METHOD M_CheckGCodeStart : ERRORID
VAR_INPUT
END_VAR
IF NOT (P_bIsInit AND pDiluter^.P_bIsInit) THEN
	M_CheckGCodeStart := E_ErrorIdCmd.ERRORID_DeviceNotInitialized;
END_IF
END_METHOD

METHOD M_CheckProcDataType : BOOL
VAR_INPUT
	eProcDataType : E_ProcDataType;
END_VAR
IF eProcDataType = E_ProcDataType.PROCDATATYPE_Temp1 THEN
	M_CheckProcDataType := TRUE;
END_IF
END_METHOD

METHOD M_CheckProps : ERRORID
VAR_INPUT
END_VAR
M_CheckProps := SUPER^.M_CheckProps();
IF M_CheckProps > 0 THEN
	RETURN;
END_IF
//Konfigurierte Properties checken
//zugeordneter Diuter
IF fbObjectDirectory.M_GetObjType(nDiluterObjId) <> E_ObjectType.OBJECTTYPE_Diluter THEN
	M_CheckProps := E_ErrorIdObjMgmt.ERRORID_InvalidDiluterObjId; //Error
	RETURN;
ELSE
	pDiluter := fbObjectDirectory.M_GetObjPointer(nDiluterObjId);
END_IF
END_METHOD

METHOD M_ExeAction : ERRORID
VAR_INPUT
	refActionData : REFERENCE TO ST_ActionData;	
END_VAR
IF NOT (eCurrentState = E_MachineState.MACHINESTATE_Idle OR
	eCurrentState = E_MachineState.MACHINESTATE_Active OR
	eCurrentState = E_MachineState.MACHINESTATE_Ready) THEN
	M_ExeAction := E_ErrorIdCmd.ERRORID_InvalidState;
	RETURN;
END_IF

CASE refActionData.eAction OF
	
	E_Action.ACTION_Init:
		IF NOT bInitAxis AND NOT bInitTool THEN
			bInitAxis := TRUE;
			bInitTool := TRUE;
			fbList.A_AddHeadValue( hList := hList, putValue := E_Action.ACTION_Init);	//InitBase
			fbList.A_AddHeadValue( hList := hList, putValue := E_Action.ACTION_Init);	//InitSpec
		ELSE
			RETURN;
		END_IF		
	
	E_Action.ACTION_Heating:
		IF nStateA_Heating = 0 THEN
			nTempSetpoint := DINT_TO_UINT(refActionData.aParams[1]);
			IF nTempSetpoint > 1000 THEN
				M_ExeAction := E_ErrorIdCmd.ERRORID_InvalidHeatingTemp;  //Error
				RETURN;
			END_IF
			bHeatingOn := DINT_TO_BOOL(refActionData.aParams[2]);			
			bHeating := TRUE;
			fbList.A_AddHeadValue(hList := hList, putValue := E_Action.ACTION_Heating);
		ELSE
			RETURN;
		END_IF		
		
	E_Action.ACTION_Aspirate:
		IF NOT bAspirate THEN
			M_ExeAction := pDiluter^.M_CheckBottles(0); //Checken, ob Bottles OK
			IF M_ExeAction > 0 THEN
				RETURN;
			END_IF
			nQuantity := refActionData.aParams[1];
			nFlow := refActionData.aParams[2];
			fbList.A_AddHeadValue( hList := hList, putValue := E_Action.ACTION_Aspirate);
			bAspirate := TRUE;
		END_IF
		
	E_Action.ACTION_Dispense:
		IF NOT bDispense THEN
			M_ExeAction := pDiluter^.M_CheckBottles(0); //Checken, ob Bottles OK
			IF M_ExeAction > 0 THEN
				RETURN;
			END_IF
			nQuantity := refActionData.aParams[1];
			nFlow := refActionData.aParams[2];
			fbList.A_AddHeadValue( hList := hList, putValue := E_Action.ACTION_Dispense);
			bDispense := TRUE;
		END_IF
		
	E_Action.ACTION_DispenseDrops:
		bDispensePiezoStart := DINT_TO_BOOL(refActionData.aParams[2]);
		IF NOT bDispensePiezo AND bDispensePiezoStart THEN
			fbPiezoControl.P_nDrops := nDrops := DINT_TO_UINT(refActionData.aParams[1]);
			fbPiezoControl.P_bStroboscope := DINT_TO_BOOL(refActionData.aParams[3]);
			bSkipValveMove := DINT_TO_BOOL(refActionData.aParams[5]);
			fbList.A_AddHeadValue(hList := hList, putValue := E_Action.ACTION_DispenseDrops);
			bDispensePiezo := TRUE;
		ELSE
			fbPiezoControl.M_StartStop(bDispensePiezoStart); //Stoppen
		END_IF
		
	E_Action.ACTION_DilMoveValve:
		//Darf nur ausgeführt werden, wenn kein Dispensen aktiv ist
		IF NOT (bAspirate OR bDispense OR bDispensePiezo OR bDilMoveValve) THEN
			M_ExeAction := pDiluter^.M_ExeAction(refActionData);
			IF M_ExeAction > 0 THEN
				RETURN;
			END_IF
			fbList.A_AddHeadValue(hList := hList, putValue := E_Action.ACTION_DilMoveValve);
			bDilMoveValve := TRUE;
		END_IF
		
	E_Action.ACTION_MoveX,E_Action.ACTION_MoveY,E_Action.ACTION_MoveXY:
		IF pZAxisRef^.stInput.nToolState.1 THEN	//ZSensor ist montiert
			M_ExeAction := ERRORID_PipMoveWithZSensor;  //Error
			RETURN;
		ELSE
			M_ExeAction := SUPER^.M_ExeAction(refActionData);
			RETURN;
		END_IF

	E_Action.ACTION_MoveZ:
		IF pZAxisRef^.stInput.nToolState.1 THEN //ZSensor ist montiert
			eMoveModeZ := DINT_TO_USINT(refActionData.aParams[1]);
			IF NOT(eMoveModeZ = E_MoveMode.MODE_Free OR eMoveModeZ = E_MoveMode.MODE_Home) THEN
				M_ExeAction := ERRORID_PipMoveWithZSensor;  //Error
				RETURN;
			END_IF
			M_ExeAction := SUPER^.M_ExeAction(refActionData);
			RETURN;			
		ELSE
			M_ExeAction := SUPER^.M_ExeAction(refActionData);
			RETURN;
		END_IF
	ELSE
		M_ExeAction := SUPER^.M_ExeAction(refActionData);
		RETURN;
END_CASE
bBusy := TRUE;
eCurrentState := E_MachineState.MACHINESTATE_Active;
END_METHOD

METHOD M_GetAllProps : ERRORID
VAR_INPUT
	refCmdData : REFERENCE TO  ST_CmdData;
END_VAR
//BaseProperties lesen
SUPER^.M_GetAllProps(refCmdData);
nCurrentPropIndex := nCurrentPropIndex + 1;
refCmdData.n32Data[nCurrentPropIndex] := P_nObjIdDiluter;
nCurrentPropIndex := nCurrentPropIndex + 1;
refCmdData.n32Data[nCurrentPropIndex] := fbPiezoControl.P_nFrequency;
nCurrentPropIndex := nCurrentPropIndex + 1;
refCmdData.n32Data[nCurrentPropIndex] := fbPiezoControl.P_nPulse;
nCurrentPropIndex := nCurrentPropIndex + 1;
refCmdData.n32Data[nCurrentPropIndex] := fbPiezoControl.P_nVoltage;
nCurrentPropIndex := nCurrentPropIndex + 1;
refCmdData.n32Data[nCurrentPropIndex] := nDrypadArea;
nCurrentPropIndex := nCurrentPropIndex + 1;
refCmdData.n32Data[nCurrentPropIndex] := TIME_TO_DINT(tDryTime);
nCurrentPropIndex := nCurrentPropIndex + 1;
IF pFbHeaterRef > 0 THEN
	refCmdData.n32Data[nCurrentPropIndex] := 1;
ELSE
	refCmdData.n32Data[nCurrentPropIndex] := 0;
END_IF
END_METHOD

METHOD M_GetProcData : DINT
VAR_INPUT
	eProcDataType : E_ProcDataType;
END_VAR
IF eProcDataType = E_ProcDataType.PROCDATATYPE_Temp1 THEN
	M_GetProcData := pFbHeaterRef^.nTemp1Actual;
END_IF
END_METHOD

METHOD M_SetAllProps : ERRORID
VAR_INPUT
	refCmdData : REFERENCE TO  ST_CmdData;
END_VAR

VAR
	pSinglePiezoHolder : POINTER TO FB_SingelPiezoHolder;
	pTwinPiezoHolder :  POINTER TO FB_TwinPiezoHolder;
END_VAR
M_SetAllProps := SUPER^.M_SetAllProps(refCmdData);

IF M_SetAllProps > 0 THEN
	RETURN;
END_IF

IF pParentMzTool^.P_eObjectType = E_ObjectType.OBJECTTYPE_SinglePiezoHolder THEN
	pSinglePiezoHolder := pParentMzTool;
	pFbPiezoRef := pSinglePiezoHolder^.M_GetPiezoRef(pParentSlot);	
ELSIF pParentMzTool^.P_eObjectType = E_ObjectType.OBJECTTYPE_TwinPiezoHolder THEN
	pTwinPiezoHolder := pParentMzTool;
	pFbPiezoRef := pTwinPiezoHolder^.M_GetPiezoRef(pParentSlot);
ELSE
	M_SetAllProps := E_ErrorIdObjMgmt.ERRORID_InvalidParentMzTool;
	RETURN;
END_IF

IF pFbPiezoRef = 0 THEN
	M_SetAllProps := E_ErrorIdObjMgmt.ERRORID_InvalidPiezoRef;
	RETURN;
END_IF

fbPiezoControl(pFbPiezoRef:= pFbPiezoRef);	//Setzt den Zeiger "pFbPiezoRef" innerhalb von fbMultiZPiezo

//Diluter
nCurrentPropIndex := nCurrentPropIndex + 1;
nSpecPropIndex := nCurrentPropIndex;
nDiluterObjId :=  DINT_TO_UINT(refCmdData.n32Data[nCurrentPropIndex]);
IF fbObjectDirectory.M_GetObjType(nDiluterObjId) = E_ObjectType.OBJECTTYPE_Diluter THEN
	pDiluter := fbObjectDirectory.M_GetObjPointer(nDiluterObjId);
ELSE
	M_SetAllProps := E_ErrorIdObjMgmt.ERRORID_InvalidDiluterObjId;
	RETURN;
END_IF

//Frequenz
nCurrentPropIndex := nCurrentPropIndex + 1;
M_SetAllProps := M_SetFrequency(refCmdData.n32Data[nCurrentPropIndex], FALSE);
IF M_SetAllProps > 0 THEN
	RETURN;
END_IF

//Plusbreite
nCurrentPropIndex := nCurrentPropIndex + 1;
M_SetAllProps := M_SetPulse(refCmdData.n32Data[nCurrentPropIndex], FALSE);
IF M_SetAllProps > 0 THEN
	RETURN;
END_IF

//Spannung
nCurrentPropIndex := nCurrentPropIndex + 1;
M_SetAllProps := M_SetVoltage(refCmdData.n32Data[nCurrentPropIndex], FALSE);
IF M_SetAllProps > 0 THEN
	RETURN;
END_IF

//DrypadArea
nCurrentPropIndex := nCurrentPropIndex + 1;
nDrypadArea := DINT_TO_USINT(refCmdData.n32Data[nCurrentPropIndex]);
IF NOT (nDrypadArea > 0 AND nDrypadArea < 3) THEN
	M_SetAllProps := E_ErrorIdObjMgmt.ERRORID_InvalidDrypadArea;
	RETURN;
END_IF

//DryTime
nCurrentPropIndex := nCurrentPropIndex + 1;
tDryTime := DINT_TO_TIME(refCmdData.n32Data[nCurrentPropIndex]);

//HeaterExist
nCurrentPropIndex := nCurrentPropIndex + 1;
pFbHeaterRef := ADR(pFbMultiZ^.aFbHeaterRef[pFbPiezoRef^.nChannel]);
IF refCmdData.n32Data[nCurrentPropIndex] = 1 THEN
	pFbHeaterRef^.P_bHeaterFixed := TRUE;
ELSE
	pFbHeaterRef^.P_bHeaterFixed := FALSE;
	pFbHeaterRef := 0;
END_IF

nNoOfProps := nCurrentPropIndex + 1;
END_METHOD

METHOD M_SetFrequency : ERRORID
VAR_INPUT
	nValue 				: DINT;
	bSetObjectChange 	: BOOL;
END_VAR
IF nValue >= 16 AND nValue < 10000 THEN
	fbPiezoControl.P_nFrequency := DINT_TO_UINT(nValue);
	IF bSetObjectChange THEN
		fbObjectDirectory.M_SetObjChange(nObjectId);
	END_IF
ELSE
	M_SetFrequency := E_ErrorIdObjMgmt.ERRORID_InvalidFrequency;
END_IF
END_METHOD

METHOD M_SetPrintParams : ST_MethResult
VAR_INPUT
	eType 		: E_PrintParamType;
	nNumerator	: USINT;
	nValue		: DINT;
END_VAR
IF nNumerator <> 1 THEN
	M_SetPrintParams.bError := TRUE;
	M_SetPrintParams.nErrorId := E_ErrorIdCmd.ERRORID_InvalidPrintParamNumerator;
	RETURN;
END_IF

CASE eType OF
	E_PrintParamType.Frequency:
		M_SetPrintParams.nErrorId := M_SetFrequency(nValue, TRUE);
	E_PrintParamType.Pulse:
		M_SetPrintParams.nErrorId := M_SetPulse(nValue, TRUE);
	E_PrintParamType.Voltage:
		M_SetPrintParams.nErrorId := M_SetVoltage(nValue, TRUE);
ELSE
	M_SetPrintParams.bError := TRUE;
	M_SetPrintParams.nErrorId := E_ErrorIdCmd.ERRORID_InvalidPrintParamType;
END_CASE

IF M_SetPrintParams.nErrorId > 0 THEN
	M_SetPrintParams.bError := TRUE;
END_IF
END_METHOD

METHOD M_SetPulse : ERRORID
VAR_INPUT
	nValue 				: DINT;
	bSetObjectChange 	: BOOL;
END_VAR
IF nValue > 0 AND nValue < 501 THEN
	fbPiezoControl.P_nPulse := DINT_TO_UINT(nValue);
	IF bSetObjectChange THEN
		fbObjectDirectory.M_SetObjChange(nObjectId);
	END_IF	
ELSE
	M_SetPulse := E_ErrorIdObjMgmt.ERRORID_InvalidPulseWidth;
END_IF
END_METHOD

METHOD M_SetSingleProp : ERRORID
VAR_INPUT
	refCmdData : REFERENCE TO  ST_CmdData;
END_VAR
IF nSpecPropIndex = refCmdData.aHeader[1] THEN
	//Diluter Id sollte nicht einzeln geändert werden können!
	M_SetSingleProp := E_ErrorIdCmd.ERRORID_InvalidProperty;	
ELSIF (nSpecPropIndex + 1) = refCmdData.aHeader[1] THEN	//Frequenz
	M_SetSingleProp := M_SetFrequency(refCmdData.n32Data[0], FALSE);
ELSIF (nSpecPropIndex + 2) = refCmdData.aHeader[1] THEN //Pulsbreite
	M_SetSingleProp := M_SetPulse(refCmdData.n32Data[0], FALSE);
ELSIF (nSpecPropIndex + 3) = refCmdData.aHeader[1] THEN	//Spannung
	M_SetSingleProp := M_SetVoltage(refCmdData.n32Data[0], FALSE);
ELSIF (nSpecPropIndex + 4) = refCmdData.aHeader[1] THEN
	IF NOT (refCmdData.n32Data[0] > 0 AND refCmdData.n32Data[0] < 3) THEN //DrypadArea
		M_SetSingleProp := E_ErrorIdObjMgmt.ERRORID_InvalidDrypadArea;
		RETURN;
	END_IF
	nDrypadArea := DINT_TO_USINT(refCmdData.n32Data[0]);
ELSIF (nSpecPropIndex + 5) = refCmdData.aHeader[1] THEN //DryTime
	tDryTime := DINT_TO_TIME(refCmdData.n32Data[0]);
ELSE
	M_SetSingleProp := SUPER^.M_SetSingleProp(refCmdData);
END_IF
END_METHOD

METHOD M_SetVoltage : ERRORID
VAR_INPUT
	nValue 				: DINT;
	bSetObjectChange 	: BOOL;
END_VAR
IF nValue > 0 AND nValue < 151 THEN
	fbPiezoControl.P_nVoltage := DINT_TO_UINT(nValue);
	IF bSetObjectChange THEN
		fbObjectDirectory.M_SetObjChange(nObjectId);
	END_IF	
ELSE
	M_SetVoltage := E_ErrorIdObjMgmt.ERRORID_InvalidVoltage;
END_IF
END_METHOD

METHOD M_StartUniDispense : ERRORID
VAR_INPUT
	nParam1 : DINT; //Drops
	nParam2 : DINT; //nicht benutzt
END_VAR

VAR_OUTPUT
	bIsContinous : BOOL;
END_VAR

VAR
	stActionData : ST_ActionData;
END_VAR
IF nParam1 = 0 THEN //DauerDispensen
	bIsContinous := TRUE;
	stActionData.aParams[1] := 0; //Continous
ELSE
	stActionData.aParams[1] := nParam1; //Drops
END_IF

stActionData.eAction := E_Action.ACTION_DispenseDrops;
stActionData.aParams[2] := 1; //On
M_StartUniDispense := M_ExeAction(stActionData);
END_METHOD

METHOD M_StopUniDispense : ERRORID
VAR_INPUT
END_VAR
M_CancelAction(E_Action.ACTION_DispenseDrops);
END_METHOD

PROPERTY P_bSensorMounted : BOOL
GET
IF pParentMzTool^.P_eObjectType = E_ObjectType.OBJECTTYPE_SinglePiezoHolder THEN
	P_bSensorMounted := pZAxisRef^.stInput.nToolState.1;	
END_IF
END_GET
END_PROPERTY

PROPERTY P_nDrypadArea : USINT
GET
P_nDrypadArea := nDrypadArea;
END_GET
END_PROPERTY

PROPERTY P_nObjIdDiluter : UINT
GET
IF pDiluter > 0 THEN
	P_nObjIdDiluter := pDiluter^.P_nObjectID;
END_IF
END_GET
END_PROPERTY

PROPERTY P_nTestResult : UDINT
GET
P_nTestResult := nTestResult;
END_GET
SET
nTestResult := P_nTestResult;
END_SET
END_PROPERTY

PROPERTY P_pDiluter : POINTER TO FB_Diluter
GET
P_pDiluter := pDiluter;
END_GET
END_PROPERTY

PROPERTY P_pPiezoRef : POINTER TO FB_PiezoRef
GET
P_pPiezoRef := pFbPiezoRef;
END_GET
END_PROPERTY

PROPERTY P_rToolRadius : REAL
GET
VAR
	stDim : ST_3DDimension;
END_VAR
P_rToolRadius := 1500.0;
END_GET
END_PROPERTY

PROPERTY P_stCurrentXYArea : FB_RectAngle
GET
VAR
	stPoint : ST_3DPoint;
END_VAR
stPoint := P_stCurrentPosPhys;
P_stCurrentXYArea.X1 := stPoint.X - 1000.0;
P_stCurrentXYArea.X2 := stPoint.X + 1000.0;
P_stCurrentXYArea.Y1 := stPoint.Y - 1000.0;
P_stCurrentXYArea.Y2 := stPoint.Y + 1000.0;
END_GET
END_PROPERTY

PROPERTY P_tDryTime : TIME
GET
P_tDryTime := tDryTime;
END_GET
END_PROPERTY

END_FUNCTION_BLOCK

// ---- Hardware/MultiZ/Piezo/FB_PiezoControl.TcPOU
FUNCTION_BLOCK FB_PiezoControl

VAR_OUTPUT
	bBusy : BOOL;
	bError : BOOL;
	nErrorId : ERRORID;
END_VAR

VAR_IN_OUT
	pFbPiezoRef	: POINTER TO FB_PiezoRef;
END_VAR

VAR
	nCyclCnt : UINT;
	nPeriodSum : UDINT;
	bLost	: BOOL;
	fbSdoWrite	: FB_SDO_WRITE;
	bSendPeriod : BOOL;
	bSendPeriodFlag : BOOL := TRUE;
	bSendPulse : BOOL;
	bSendPulseFlag : BOOL := TRUE;
	bSendVoltage : BOOL;
	bSendVoltageFlag : BOOL := TRUE;
	bSendHoldVoltage : BOOL;
	bSendHoldVoltageFlag : BOOL := TRUE;
	bSendPrePeakTime : BOOL;
	bSendPrePeakTimeFlag : BOOL := TRUE;
	bSendDrops : BOOL;
	bSendDropsFlag : BOOL := TRUE;
	bStroboscope : BOOL;
	fbFTrig : F_TRIG;
END_VAR

IF pFbPiezoRef = 0 THEN
	RETURN;
END_IF

IF bSendPeriod THEN
	IF bSendPeriodFlag XOR fbSdoWrite.bBusy THEN
		bSendPeriodFlag := FALSE;
		fbSdoWrite(sADSNetID:= pFbPiezoRef^.pMultiZRef^.P_sAdsNetId, nPortNr:= pFbPiezoRef^.pMultiZRef^.P_nAdsPort,
					nIndex:= cPiezoPeriod.nIndex, nSubIndex:= pFbPiezoRef^.nChannel, 
					nDataLength:= cPiezoPeriod.nLength, nData:= pFbPiezoRef^.P_nPeriod, bExecute:= TRUE);
	END_IF

	IF NOT fbSdoWrite.bBusy THEN
		IF fbSdoWrite.bError THEN
			bError := TRUE;
			nErrorId := fbSdoWrite.nAdsErrorId;
		END_IF
		fbSdoWrite(bExecute:= FALSE);
		bSendPeriodFlag := TRUE;
		bSendPeriod := FALSE;
	END_IF	
END_IF	

IF bSendPulse THEN
	IF bSendPulseFlag XOR fbSdoWrite.bBusy THEN
		bSendPulseFlag := FALSE;
		fbSdoWrite(sADSNetID:= pFbPiezoRef^.pMultiZRef^.P_sAdsNetId, nPortNr:= pFbPiezoRef^.pMultiZRef^.P_nAdsPort,
					nIndex:= cPiezoPulse.nIndex, nSubIndex:= pFbPiezoRef^.nChannel, 
					nDataLength:= cPiezoPulse.nLength, nData:= pFbPiezoRef^.P_nPulse, bExecute:= TRUE);
	END_IF
	IF NOT fbSdoWrite.bBusy THEN
		IF fbSdoWrite.bError THEN
			bError := TRUE;
			nErrorId := fbSdoWrite.nAdsErrorId;
		END_IF
		fbSdoWrite(bExecute:= FALSE);
		bSendPulseFlag := TRUE;
		bSendPulse := FALSE;
	END_IF
END_IF	

IF bSendVoltage THEN
	IF bSendVoltageFlag XOR fbSdoWrite.bBusy THEN
		bSendVoltageFlag := FALSE;
		fbSdoWrite(sADSNetID:= pFbPiezoRef^.pMultiZRef^.P_sAdsNetId, nPortNr:= pFbPiezoRef^.pMultiZRef^.P_nAdsPort,
					nIndex:= cPiezoVoltage.nIndex, nSubIndex:= pFbPiezoRef^.nChannel, 
					nDataLength:= cPiezoVoltage.nLength, nData:= pFbPiezoRef^.P_nVoltage, bExecute:= TRUE);
	END_IF
	IF NOT fbSdoWrite.bBusy THEN
		IF fbSdoWrite.bError THEN
			bError := TRUE;
			nErrorId := fbSdoWrite.nAdsErrorId;
		END_IF
		fbSdoWrite(bExecute:= FALSE);
		bSendVoltageFlag := TRUE;
		bSendVoltage := FALSE;
	END_IF
END_IF

IF bSendHoldVoltage THEN
	IF bSendHoldVoltageFlag XOR fbSdoWrite.bBusy THEN
		bSendHoldVoltageFlag := FALSE;
		fbSdoWrite(sADSNetID:= pFbPiezoRef^.pMultiZRef^.P_sAdsNetId, nPortNr:= pFbPiezoRef^.pMultiZRef^.P_nAdsPort,
					nIndex:= cPiezoHoldVoltage.nIndex, nSubIndex:= pFbPiezoRef^.nChannel, 
					nDataLength:= cPiezoHoldVoltage.nLength, nData:= pFbPiezoRef^.P_nHoldVoltage, bExecute:= TRUE);
	END_IF
	IF NOT fbSdoWrite.bBusy THEN
		IF fbSdoWrite.bError THEN
			bError := TRUE;
			nErrorId := fbSdoWrite.nAdsErrorId;
		END_IF
		fbSdoWrite(bExecute:= FALSE);
		bSendHoldVoltageFlag := TRUE;
		bSendHoldVoltage := FALSE;
	END_IF
END_IF

IF bSendPrePeakTime THEN
	IF bSendPrePeakTimeFlag XOR fbSdoWrite.bBusy THEN
		bSendPrePeakTimeFlag := FALSE;
		fbSdoWrite(sADSNetID:= pFbPiezoRef^.pMultiZRef^.P_sAdsNetId, nPortNr:= pFbPiezoRef^.pMultiZRef^.P_nAdsPort,
					nIndex:= cPiezoPrePeakTime.nIndex, nSubIndex:= pFbPiezoRef^.nChannel, 
					nDataLength:= cPiezoPrePeakTime.nLength, nData:= pFbPiezoRef^.P_nPrePeakTime, bExecute:= TRUE);
	END_IF
	IF NOT fbSdoWrite.bBusy THEN
		IF fbSdoWrite.bError THEN
			bError := TRUE;
			nErrorId := fbSdoWrite.nAdsErrorId;
		END_IF
		fbSdoWrite(bExecute:= FALSE);
		bSendPrePeakTimeFlag := TRUE;
		bSendPrePeakTime := FALSE;
	END_IF
END_IF

IF bSendDrops THEN
	IF bSendDropsFlag XOR fbSdoWrite.bBusy THEN
		bSendDropsFlag := FALSE;
		fbSdoWrite(sADSNetID:= pFbPiezoRef^.pMultiZRef^.P_sAdsNetId, nPortNr:= pFbPiezoRef^.pMultiZRef^.P_nAdsPort,
					nIndex:= cPiezoDrops.nIndex, nSubIndex:= pFbPiezoRef^.nChannel, 
					nDataLength:= cPiezoDrops.nLength, nData:= pFbPiezoRef^.P_nDrops, bExecute:= TRUE);
	END_IF
	IF NOT fbSdoWrite.bBusy THEN
		IF fbSdoWrite.bError THEN
			bError := TRUE;
			nErrorId := fbSdoWrite.nAdsErrorId;
		END_IF
		fbSdoWrite(bExecute:= FALSE);
		bSendDropsFlag := TRUE;
		bSendDrops := FALSE;
	END_IF
END_IF

{warning 'siehe Kommentar'}
//wurde gegeüber Version V2.0.16.X überarbeitet und ist noch nicht im Dauertest gelaufen
//es ist nicht ausgeschlossen, dass wenn das ToolState nicht "1" wird, dieser Baustein immer im Busy bleibt, da nur auf eine fallende Flanke reagiert wird

//Für den Fall, dass die Anzahl der Tropfen x Periodendauer 20ms unterschreitet, kann es dazu führen, dass das Statusbit nicht erfasst werden kann. Das hängt
//stark von der Laufzeit der Kopfbasis ab. In diesem Fall sollte 
//Man könnte auch davon ausgehen, dass spätestens im zweiten Zyklus nach dem bBusy auf true gewechselt hat, der Toolstate entsprechend auf true wechselt
//Wenn das nicht der Fall ist, dann überprüfen, ob Periodendauer x Zykluszeit kleiner 20ms.

IF bBusy THEN
	fbFTrig(CLK:= pFbPiezoRef^.pToolState^.0); 
	IF fbFTrig.Q THEN
		pFbPiezoRef^.pToolCtrl^.0 := FALSE;
		pFbPiezoRef^.pToolCtrl^.1 := FALSE;
		pFbPiezoRef^.P_bSynchronize := FALSE;
		bBusy := FALSE;
	END_IF
	IF bBusy THEN
		nCyclCnt := nCyclCnt + 1;
		IF nCyclCnt = 4 THEN
			//Hier sollte spätestens der ToolState auf 1 gesetzt sein
			IF NOT pFbPiezoRef^.pToolState^.0 THEN
				bLost := TRUE;
				nPeriodSum := pFbPiezoRef^.P_nPeriod * pFbPiezoRef^.P_nDrops;
				IF (pFbPiezoRef^.P_nDrops > 0) AND  (nPeriodSum < 20000) THEN
					//der ToolState wurde wahrscheinlich verpasst
					pFbPiezoRef^.pToolCtrl^.0 := FALSE;
					pFbPiezoRef^.pToolCtrl^.1 := FALSE;
					pFbPiezoRef^.P_bSynchronize := FALSE;
					bBusy := FALSE;
				END_IF
			END_IF
		END_IF
	END_IF
END_IF

METHOD M_Init : ERRORID
VAR_INPUT
END_VAR

VAR
	nMode	: BYTE;
END_VAR
IF NOT pFbPiezoRef^.pMultiZRef^.P_bLegacy THEN
	nMode := pFbPiezoRef^.P_eDispenserMode;
	nMode := SHL(nMode,3);
	pFbPiezoRef^.pToolCtrl^ := pFbPiezoRef^.pToolCtrl^ OR nMode;	
	bSendHoldVoltage := TRUE;
	bSendPrePeakTime := TRUE;
END_IF
bSendPeriod := TRUE;
bSendPulse := TRUE;
bSendVoltage := TRUE;
END_METHOD

METHOD M_StartStop
VAR_INPUT
	bStart : BOOL;
END_VAR
IF bStart THEN
	IF NOT bBusy THEN
		nCyclCnt := 0;
		bBusy := TRUE;
		bLost := FALSE;
	END_IF
	pFbPiezoRef^.pToolCtrl^.0 := TRUE;
	pFbPiezoRef^.pToolCtrl^.1 := bStroboscope;
	pFbPiezoRef^.pToolCtrl^.2 := TRUE; //LED am Pipettenhalter
	pFbPiezoRef^.pToolCtrl^.5 := pFbPiezoRef^.P_bSynchronize;
ELSE
	pFbPiezoRef^.pToolCtrl^.0 := FALSE;
	pFbPiezoRef^.pToolCtrl^.1 := FALSE;
	pFbPiezoRef^.pToolCtrl^.2 := FALSE; //LED am Pipettenhalter
	pFbPiezoRef^.pToolCtrl^.5 := FALSE; //Synchronize
END_IF
END_METHOD

PROPERTY P_bIsSending : BOOL
GET
P_bIsSending := bSendPeriod OR bSendPulse OR bSendVoltage OR bSendHoldVoltage OR bSendPrePeakTime OR bSendDrops;
END_GET
END_PROPERTY

PROPERTY P_bStroboscope : BOOL
SET
bStroboscope := P_bStroboscope;
pFbPiezoRef^.pToolCtrl^.1 := bStroboscope;
END_SET
END_PROPERTY

PROPERTY P_nDrops : UINT
GET
IF pFbPiezoRef > 0 THEN
	P_nDrops := pFbPiezoRef^.P_nDrops;
END_IF
END_GET
SET
IF pFbPiezoRef > 0 THEN
	IF P_nDrops <> pFbPiezoRef^.P_nDrops THEN
		pFbPiezoRef^.P_nDrops := P_nDrops;
		bSendDrops := TRUE;
	END_IF
END_IF
END_SET
END_PROPERTY

PROPERTY P_nFrequency : UINT
GET
IF pFbPiezoRef > 0 THEN
	IF pFbPiezoRef^.P_nPeriod <> 0 THEN
		P_nFrequency := UDINT_TO_UINT(1000000 / pFbPiezoRef^.P_nPeriod);
	ELSE
		P_nFrequency := 0;	
	END_IF
END_IF
END_GET
SET
VAR
	nPeriodTemp : UINT;
END_VAR
IF pFbPiezoRef > 0 THEN
	nPeriodTemp := UDINT_TO_UINT(1000000/P_nFrequency);
	IF nPeriodTemp <> pFbPiezoRef^.P_nPeriod THEN
		pFbPiezoRef^.P_nPeriod := nPeriodTemp;
		bSendPeriod := TRUE;
	END_IF	
END_IF
END_SET
END_PROPERTY

PROPERTY P_nHoldVoltage : UINT
GET
IF pFbPiezoRef > 0 THEN
	P_nHoldVoltage := pFbPiezoRef^.P_nHoldVoltage;
END_IF
END_GET
SET
IF pFbPiezoRef > 0 THEN
	IF P_nHoldVoltage <> pFbPiezoRef^.P_nHoldVoltage THEN
		pFbPiezoRef^.P_nHoldVoltage := P_nHoldVoltage;
		bSendHoldVoltage := TRUE;
	END_IF
END_IF
END_SET
END_PROPERTY

PROPERTY P_nPrePeakTime : UINT
GET
IF pFbPiezoRef > 0 THEN
	P_nPrePeakTime := pFbPiezoRef^.P_nPrePeakTime;
END_IF
END_GET
SET
IF pFbPiezoRef > 0 THEN
	IF P_nPrePeakTime <> pFbPiezoRef^.P_nPrePeakTime THEN
		pFbPiezoRef^.P_nPrePeakTime := P_nPrePeakTime;
		bSendPrePeakTime := TRUE;
	END_IF
END_IF
END_SET
END_PROPERTY

PROPERTY P_nPulse : UINT
GET
IF pFbPiezoRef > 0 THEN
	P_nPulse := pFbPiezoRef^.P_nPulse;
END_IF
END_GET
SET
IF pFbPiezoRef > 0 THEN
	IF P_nPulse <> pFbPiezoRef^.P_nPulse THEN
		pFbPiezoRef^.P_nPulse := P_nPulse;
		bSendPulse := TRUE;
	END_IF
END_IF
END_SET
END_PROPERTY

PROPERTY P_nVoltage : UINT
GET
IF pFbPiezoRef > 0 THEN
	P_nVoltage := pFbPiezoRef^.P_nVoltage;
END_IF
END_GET
SET
IF pFbPiezoRef > 0 THEN
	IF P_nVoltage <> pFbPiezoRef^.P_nVoltage THEN
		pFbPiezoRef^.P_nVoltage := P_nVoltage;
		bSendVoltage := TRUE;
	END_IF
END_IF
END_SET
END_PROPERTY

END_FUNCTION_BLOCK

// ---- Objects/Tools/FB_SingelPiezoHolder.TcPOU
FUNCTION_BLOCK FB_SingelPiezoHolder EXTENDS FB_MzTool
VAR_INPUT
END_VAR
VAR_OUTPUT
END_VAR
VAR
	//SpecProperties
	//****************************************Aktionvariablen****************************************************
	
END_VAR

IF eCurrentState = E_MachineState.MACHINESTATE_Active THEN
	;

END_IF

SUPER^();	//FB_MzTool aufrufen

//Prozessdaten aktualisieren

aObjProcData[nNotifyId] := stProcessData;

ACTION A_Reset:
IF nStateA_ResetSpec = 0 THEN 
	nStateA_ResetSpec := 80;		
END_IF

SUPER^.A_Reset();
END_ACTION

ACTION A_Stop:
IF nStateA_Stop = 0 THEN
	nStateA_Stop := 1;
END_IF

SUPER^.A_Stop();
END_ACTION

METHOD FB_init : BOOL
VAR_INPUT
	bInitRetains : BOOL; // if TRUE, the retain variables are initialized (warm start / cold start)
	bInCopyCode : BOOL;  // if TRUE, the instance afterwards gets moved into the copy code (online change)
END_VAR
eObjectType := E_ObjectType.OBJECTTYPE_SinglePiezoHolder;
eObjectGroup := E_ObjectGroup.OBJECTGROUP_MzTool OR E_ObjectGroup.OBJECTGROUP_Device;
END_METHOD

METHOD M_AddChild : ERRORID
VAR_INPUT
	pObject : POINTER TO FB_Object;
	nSlotNr	: UINT;
	nIndex 	: INT;
END_VAR
//Kann folgende Objekt-Typen aufnehmen
//ZSensor, Piezo, PassivPip, Solenoid
IF pObject > 0 THEN
	IF pObject^.P_eObjectType = E_ObjectType.OBJECTTYPE_ZSensor OR
		pObject^.P_eObjectType = E_ObjectType.OBJECTTYPE_PiezoPip OR
		pObject^.P_eObjectType = E_ObjectType.OBJECTTYPE_PassivPip OR
		pObject^.P_eObjectType = E_ObjectType.OBJECTTYPE_DummyTool OR
		pObject^.P_eObjectType = E_ObjectType.OBJECTTYPE_Camera OR
		pObject^.P_eObjectType = E_ObjectType.OBJECTTYPE_SolenoidPip THEN
		M_AddChild := SUPER^.M_AddChild(pObject,nSlotNr,nIndex);
	ELSE
		M_AddChild := E_ErrorIdObjMgmt.ERRORID_InvalidParentObject;
	END_IF
ELSE
	M_AddChild := E_ErrorIdObjMgmt.ERRORID_InvalidParentObject;
END_IF
END_METHOD

METHOD M_CheckAction : ERRORID
VAR_INPUT
	refActionData 	: REFERENCE TO ST_ActionData;
	pCorrelObject	: POINTER TO FB_Object;
END_VAR

VAR
END_VAR
CASE refActionData.eAction OF
	E_Action.ACTION_ActionOnArray,
	E_Action.ACTION_MoveToTarget:
		M_CheckAction := E_ErrorIdCmd.ERRORID_InvalidAction; //würde sonst durch Base erlaubt werden
ELSE
	M_CheckAction := SUPER^.M_CheckAction(refActionData, pCorrelObject);
END_CASE
END_METHOD

METHOD M_ExeAction : ERRORID
VAR_INPUT
	refActionData : REFERENCE TO ST_ActionData;	
END_VAR
IF NOT (eCurrentState = E_MachineState.MACHINESTATE_Idle OR
	eCurrentState = E_MachineState.MACHINESTATE_Active OR
	eCurrentState = E_MachineState.MACHINESTATE_Ready) THEN
	M_ExeAction := E_ErrorIdCmd.ERRORID_InvalidState;
	RETURN;
END_IF

CASE refActionData.eAction OF
	
	
	ELSE
		M_ExeAction := SUPER^.M_ExeAction(refActionData);
		RETURN;
END_CASE

bBusy := TRUE;
eCurrentState := E_MachineState.MACHINESTATE_Active;
END_METHOD

METHOD M_GetPiezoRef : POINTER TO FB_PiezoRef
VAR_INPUT
	pToolSlot	: POINTER TO FB_Slot;
END_VAR
M_GetPiezoRef := ADR(pFbMultiZ^.aFbPiezoRef[pParentSlot^.P_nNr]);
END_METHOD

METHOD M_SetAllProps : ERRORID
VAR_INPUT
	refCmdData : REFERENCE TO  ST_CmdData;
END_VAR
M_SetAllProps := SUPER^.M_SetAllProps(refCmdData);

IF M_SetAllProps > 0 THEN
	RETURN;
END_IF

pZAxisRef^.eFixedToolType := E_MzToolType.TOOL_TYPE_PiezoPip;
END_METHOD

PROPERTY P_bHasZSensorSlot : BOOL
GET
IF eObjectType = E_ObjectType.OBJECTTYPE_SinglePiezoHolder THEN
	P_bHasZSensorSlot := TRUE;	
END_IF
END_GET
END_PROPERTY

END_FUNCTION_BLOCK

// ---- GCode/FB_BuildGroup.TcPOU
FUNCTION_BLOCK FB_BuildGroup
VAR_INPUT
	bExecute	: BOOL;
END_VAR
VAR_OUTPUT
	bBusy		: BOOL;
	bError		: BOOL;
	nErrorId	: ERRORID;
END_VAR
VAR_IN_OUT
	stGCodeRef : ST_GCodeRef;
END_VAR
VAR
	nState				: USINT;
	fbCfgBuild3DGroup	: Tc2_NCI.CfgBuildExt3DGroup;
	fbMcGearIn			: Tc2_MC2.MC_GearIn;
	fbMcGearOut			: Tc2_MC2.MC_GearOut;
	pNciToPlc 			: POINTER TO NCTOPLC_NCICHANNEL_REF;
	pXDrive				: POINTER TO FB_XYDriveBase;
	pYDrive				: POINTER TO FB_XYDriveBase;
	pTwinDrive			: POINTER TO FB_XYDrive_Beck_Twin;
END_VAR

//hier werden die XYZ-Antriebe zur einer NCI-Gruppe hinzugefügt
//für den Fall, dass ein Antrieb aus zwei Motoren besteht(TwinDrive), vorher auskoppeln und danach wieder einkoppeln
IF bExecute THEN
	CASE nState OF
		0:	//X-Slave-Achse auskoppeln
			//darf nicht wie bisher über die Instanz des Drives gemacht werden, da es ab 4022.5 nicht mehrt erlaubt ist,
			//Instanzen von FBs taskübergreifend zu nutzen
			bBusy := TRUE;
			pNciToPlc := ADR(stGCodeRef.sNciToPlc);
			pXDrive := stGCodeRef.pHead^.P_pXDrive;
			pYDrive := stGCodeRef.pHead^.P_pYDrive;
			IF pXDrive^.P_bIsTwinDrive THEN
				pTwinDrive := pXDrive;
				fbMcGearOut(Slave := pTwinDrive^.P_pAxisRefSlave^, Execute:= TRUE);
				IF NOT fbMcGearOut.Busy THEN
					IF fbMcGearOut.Error THEN
						nErrorId := UDINT_TO_UINT(fbMcGearOut.ErrorID);
						nState := 99;
					ELSE
						nState := 1;
					END_IF
					fbMcGearOut(Slave := pTwinDrive^.P_pAxisRefSlave^, Execute:= FALSE);
				END_IF
			ELSE
				nState := 1;
			END_IF
			
		1:	//Interpolationsgruppe bilden
			fbCfgBuild3DGroup(bExecute:= TRUE, nGroupId:= ItpGetGroupId(pNciToPlc^),	
								nXAxisId:= pXDrive^.P_pAxisRef^.NcToPlc.AxisId,
								nYAxisId:= pYDrive^.P_pAxisRef^.NcToPlc.AxisId, 
								nQ1AxisId:= AxisRefQ1.NcToPlc.AxisId);
			IF NOT fbCfgBuild3DGroup.bBusy THEN
				IF fbCfgBuild3DGroup.bErr THEN
					nErrorId := UDINT_TO_UINT(fbCfgBuild3DGroup.nErrId);
					nState := 99;
				ELSE
					IF pXDrive^.P_bIsTwinDrive THEN
						nState := 2;
					ELSE
						bBusy := FALSE;
						nState := 80;
					END_IF
				END_IF
				fbCfgBuild3DGroup(bExecute:= FALSE);
			END_IF
		
		2:	//X-Slave-Achse ankoppeln
			fbMcGearIn(Master:= pTwinDrive^.P_pAxisRef^, Slave:= pTwinDrive^.P_pAxisRefSlave^, Execute:= TRUE, RatioNumerator:= 1.0);
			IF NOT fbMcGearIn.Busy THEN
				IF fbMcGearIn.Error THEN
					nErrorId := UDINT_TO_UINT(fbMcGearIn.ErrorID);
					nState := 99;
				ELSE
					bBusy := FALSE;
					nState := 80;
				END_IF
				fbMcGearIn(Master:= pTwinDrive^.P_pAxisRef^, Slave:= pTwinDrive^.P_pAxisRefSlave^, Execute:= FALSE);
			END_IF
	END_CASE
	
	IF nState = 99 THEN
		bError := TRUE;
		bBusy := FALSE;	
	END_IF
ELSE
	bError := FALSE;
	nErrorId := 0;
	nState := 0;
END_IF

END_FUNCTION_BLOCK

// ---- Hardware/XYDrive/FB_XYDrive_Beck_Twin.TcPOU
FUNCTION_BLOCK FB_XYDrive_Beck_Twin EXTENDS FB_XYDrive_Beck
VAR PERSISTENT
	rRefPosSlave : REAL;
END_VAR
VAR_INPUT
END_VAR
VAR_OUTPUT
END_VAR
VAR
	bHomeSwitchSlave 		AT %I* : BOOL;
	fbMcHomingSlave			: Tc2_MC2.MC_Home;
	fbMcMoveAbsSlave		: Tc2_MC2.MC_MoveAbsolute;
	fbMcHaltSlave			: Tc2_MC2.MC_Halt;
	timeout : TON;
	stMethResult			: ST_MethResult;
	bPowerOn				: BOOL;
	nStateA_PowerOn			: USINT;
	bFlag1					: BOOL;
	bFlag2					: BOOL;
	pAxisRefSlave			: POINTER TO Tc2_MC2.AXIS_REF;
	fbClearGroup			: FB_ClearGroup;
END_VAR

SUPER^();
IF bPowerOn THEN
	A_PowerOn();
	IF nStateA_PowerOn >= 80 THEN
		IF nStateA_PowerOn >= 99 THEN
			bError := TRUE;
		END_IF
		nStateA_PowerOn := 0;
		bPowerOn := FALSE;
	END_IF
END_IF
pAxisRefSlave^.ReadStatus();
bHomed := pAxisRefMaster^.Status.Homed AND pAxisRefSlave^.Status.Homed;

ACTION A_Error:
IF nStateA_Error = 0 THEN
	IF nErrorId = 17744 OR nErrorId = 18000 THEN //Schleppabstandüberwachung "Position" bzw Antriebshardware nicht bereit
		nStateA_Error := 1;
	END_IF
END_IF

CASE nStateA_Error OF
	1: //Master ausschalten
		fbMcPower(Axis:= pAxisRefMaster^, Enable:= FALSE);
		IF NOT fbMcPower.Busy THEN
			nStateA_Error := 2;
		END_IF

	2: //Slave ausschalten	
		fbMcPower(Axis:= pAxisRefSlave^, Enable:= FALSE);
		IF NOT fbMcPower.Busy THEN
			nStateA_Error := 3;
		END_IF
		
	3:	//Calibration Master + Slave zurücksetzen
		fbMcHome(Axis:= pAxisRefMaster^, Execute:= TRUE, HomingMode:= MC_ResetCalibration);
		fbMcHomingSlave(Axis:= pAxisRefSlave^, Execute:= TRUE, HomingMode:= MC_ResetCalibration);
		
		IF NOT fbMcHome.Busy AND NOT fbMcHome.Busy THEN
			IF fbMcHome.Error OR fbMcHomingSlave.Error THEN
				nStateA_Error := 99;
			ELSE
				nStateA_Error := 4;
			END_IF
			fbMcHome(Axis:= pAxisRefMaster^, Execute:= FALSE);
			fbMcHomingSlave(Axis:= pAxisRefSlave^, Execute:= FALSE);
		END_IF
END_CASE
END_ACTION

ACTION A_Init:
IF timeout.Q THEN
	nErrorId := ERRORID_SimultanErrorX1X2;
	nStateA_Init := 90;
END_IF

CASE nStateA_Init OF
	0:	//DriveAdress Masterachse ermitteln (EncoderId wird für TriggerRef benötigt)
		bBusy := TRUE;
		fbMcReadDriveAddress(Axis:= pAxisRefMaster^ ,Execute:= TRUE, DriveAddress=> stDriveAddress);
		IF NOT fbMcReadDriveAddress.Busy THEN
			IF fbMcReadDriveAddress.Error THEN
				nErrorId := UDINT_TO_UINT(fbMcReadDriveAddress.ErrorID);
				nStateA_Init := 99;
			ELSE
				stTriggerRef.EncoderID := stDriveAddress.NcEncoderId;
				IF GCode.P_bNciAvailable THEN
					nStateA_Init := 1;
				ELSE
					nStateA_Init := 2;
				END_IF
			END_IF
			fbMcReadDriveAddress(Axis:= pAxisRefMaster^ ,Execute:= FALSE);
		END_IF
		
	1:	//NCI-Gruppe auflösen ohne Slave-Achse einzukopplen
		IF GCode.bBusy OR GCode.bError THEN
			nStateA_Init := 99;
		ELSE
			fbClearGroup(bExecute:= TRUE, bReGearInSlave:= FALSE, stGCodeRef:= GCode.stGCodeRef);
			IF NOT fbClearGroup.bBusy THEN
				IF fbClearGroup.bError THEN
					nErrorId := fbClearGroup.nErrorId;
					nStateA_Init := 99;
				ELSE
					pAxisRefSlave^.ReadStatus();
					IF pAxisRefSlave^.Status.Coupled THEN
						nStateA_Init := 2;
					ELSE
						nStateA_Init := 3;
					END_IF
				END_IF
				fbClearGroup(bExecute:= FALSE, bReGearInSlave:= FALSE, stGCodeRef:= GCode.stGCodeRef);
			END_IF
		END_IF
		
	2:	//Slave auskoppeln
		stMethResult := M_GearOut();
		IF NOT stMethResult.bBusy THEN
			IF stMethResult.bError THEN
				nErrorId := stMethResult.nErrorID;
				nStateA_Init := 99;	
			ELSE
				nStateA_Init := 3;	
			END_IF
		END_IF
	
	3:	//Masterachse im Fehlerzustand?
		IF pAxisRefMaster^.Status.Error OR fbMcReset.Busy  THEN
			fbMcReset(Axis:= pAxisRefMaster^, Execute:= TRUE); 
			IF fbMcReset.Error THEN	//Error beim zurücksetzen
				nErrorId := UDINT_TO_UINT(fbMcReset.ErrorID);
				fbMcReset(Axis:= pAxisRefMaster^, Execute := FALSE);
				nStateA_Init := 99;
			ELSIF  fbMcReset.Done THEN
				fbMcReset(Axis:= pAxisRefMaster^, Execute := FALSE);
				nStateA_Init := 4;
			END_IF
		ELSE
			nStateA_Init := 4;
		END_IF
		
	4:	//Slaveachse im Fehlerzustand?
		IF pAxisRefSlave^.Status.Error OR fbMcReset.Busy THEN
			fbMcReset(Axis:= pAxisRefSlave^, Execute:= TRUE);
			IF fbMcReset.Error THEN	//Error beim zurücksetzen
				nErrorId := UDINT_TO_UINT(fbMcReset.ErrorID);
				fbMcReset(Axis:= pAxisRefSlave^, Execute := FALSE);
				nStateA_Init := 99;
			ELSIF  fbMcReset.Done THEN
				fbMcReset(Axis:= pAxisRefSlave^, Execute := FALSE);
				nStateA_Init := 5;
			END_IF
		ELSE
			nStateA_Init := 5;
		END_IF		

	5:	//Masterachse freigegeben?
		IF NOT pAxisRefMaster^.Status.ControlLoopClosed THEN
			fbMcPower(Axis:= pAxisRefMaster^, Enable:= TRUE, Enable_Positive:= TRUE, Enable_Negative:= TRUE, Override:= 100 );
			IF fbMcPower.Error THEN	 //Error bei Ausführung
				nErrorId := UDINT_TO_UINT(fbMcPower.ErrorID);
				fbMcPower(Axis:= pAxisRefMaster^, Enable:= FALSE);
				nStateA_Init := 99;
			END_IF
		ELSE
			nStateA_Init := 6;
		END_IF

	6:	//Slaveachse freigegeben?
		IF NOT pAxisRefSlave^.Status.ControlLoopClosed THEN
			fbMcPower(Axis:= pAxisRefSlave^, Enable:= TRUE, Enable_Positive:= TRUE, Enable_Negative:= TRUE, Override:= 100);
			IF fbMcPower.Error THEN	 //Error bei Ausführung
				nErrorId := UDINT_TO_UINT(fbMcPower.ErrorID);
				fbMcPower(Axis:= pAxisRefMaster^, Enable:= FALSE);
				fbMcPower(Axis:= pAxisRefSlave^, Enable:= FALSE);
				nStateA_Init := 99;
			END_IF
		ELSE
			nStateA_Init := 7;
		END_IF
		
	7:	//TouchProbe abbrechen
		fbMcAbortTrigger(Axis:= pAxisRefMaster^, TriggerInput:= stTriggerRef, Execute:= TRUE);
		IF NOT fbMcAbortTrigger.Busy THEN
			IF fbMcAbortTrigger.Error THEN
				nErrorId := UDINT_TO_UINT(fbMcAbortTrigger.ErrorID);
				nStateA_Init := 92;
			ELSE
				IF NOT bReInit AND pAxisRefMaster^.Status.Homed AND pAxisRefSlave^.Status.Homed THEN
					nStateA_Init := 10; //Slave Achse an Masterachse ankoppeln
				ELSE
					nStateA_Init := 8; //Achsen referenzieren
				END_IF
			END_IF
			fbMcAbortTrigger(Axis:= pAxisRefMaster^ ,TriggerInput:= stTriggerRef, Execute:= FALSE);
		END_IF
		
	8:	//Achsen referenzieren
		//Wenn eine Achse einen Fehler meldet, dann das Homing für die andere Achse abbrechen
		fbMcHome(Axis:= pAxisRefMaster^, Execute:= TRUE, Position:= rHomePos,
								HomingMode:= MC_DefaultHoming,	bCalibrationCam:= bHomeSwitchMaster);
							
		fbMcHomingSlave(Axis:= pAxisRefSlave^, Execute:= TRUE, Position:= rHomePosSlave,
								HomingMode:= MC_DefaultHoming, bCalibrationCam:= bHomeSwitchSlave);
							
		IF NOT fbMcHome.Busy THEN
			IF fbMcHome.Error THEN
				nErrorId := UDINT_TO_UINT(fbMcHome.ErrorID);
				fbMcHome(Axis:= pAxisRefMaster^, Execute := FALSE);
				nStateA_Init := 91;
			END_IF
		END_IF
		
		IF NOT fbMcHomingSlave.Busy THEN
			IF fbMcHomingSlave.Error THEN
				nErrorId := UDINT_TO_UINT(fbMcHomingSlave.ErrorID);
				fbMcHomingSlave(Axis:= pAxisRefSlave^, Execute := FALSE);
				nStateA_Init := 91;
			END_IF
		END_IF
		
		//Es müssen sowohl die Nocken als auch die Referenzpositionen jeweils im gleichen Zeitfenster kommen
		IF fbMcHome.Done OR fbMcHomingSlave.Done THEN
			timeout(IN:= TRUE, PT:= T#200MS);
		END_IF
		
		IF fbMcHome.Done AND fbMcHomingSlave.Done THEN
			timeout(IN:= FALSE);
			fbMcHome(Axis:= pAxisRefMaster^, Execute := FALSE);
			fbMcHomingSlave(Axis:= pAxisRefSlave^, Execute := FALSE);
			nStateA_Init := 9;
		END_IF
		
		IF bStop THEN
			nStateA_Init := 50;
		END_IF
		
	9:	//Achsen auf Durchschnitt von Referenzpunkt zurückfahren
		fbMcMoveAbs(Axis:= pAxisRefMaster^, Execute:= TRUE, Position:= (rHomePos + rHomePosSlave)/2.0 , Velocity:= 10.0);
		
		IF NOT fbMcMoveAbs.Busy THEN
			IF fbMcMoveAbs.Error	THEN
				nErrorId := UDINT_TO_UINT(fbMcMoveAbs.ErrorID);
				fbMcMoveAbs(Axis:= pAxisRefMaster^, Execute:= FALSE);
				nStateA_Init := 90;
			END_IF
		END_IF
		
		fbMcMoveAbsSlave(Axis:= pAxisRefSlave^, Execute:= TRUE, Position:= (rHomePos + rHomePosSlave)/2.0 , Velocity:= 10.0);
		
		IF NOT fbMcMoveAbsSlave.Busy THEN
			IF fbMcMoveAbsSlave.Error	THEN
				nErrorId := UDINT_TO_UINT(fbMcMoveAbsSlave.ErrorID);
				fbMcMoveAbsSlave(Axis:= pAxisRefSlave^, Execute:= FALSE);
				nStateA_Init := 90;
			END_IF
		END_IF
		
		IF fbMcMoveAbs.Done AND fbMcMoveAbsSlave.Done THEN
			fbMcMoveAbs(Axis:= pAxisRefMaster^ , Execute:= FALSE);
			fbMcMoveAbsSlave(Axis:= pAxisRefSlave^ , Execute:= FALSE);
			nStateA_Init := 10;
		END_IF
		
		IF bStop THEN
			nStateA_Init := 50;
		END_IF
		
	10:	//Slave an Master ankoppeln
		stMethResult := M_GearIn();
		IF NOT stMethResult.bBusy THEN
			IF stMethResult.bError THEN
				nErrorId := stMethResult.nErrorID;
				nStateA_Init := 92;	
			ELSE
				IF bStop THEN
					nStateA_Init := 50;
				ELSE
					nStateA_Init := 80;
				END_IF
			END_IF
		END_IF
		
	50:	//Stop
		fbMcHalt(Axis:= pAxisRefMaster^, Execute:= TRUE);
		fbMcHaltSlave(Axis:= pAxisRefSlave^, Execute:= TRUE);
		IF NOT (fbMcHalt.Busy OR fbMcHaltSlave.Busy) THEN
			fbMcHalt(Axis:= pAxisRefMaster^, Execute:= FALSE);
			fbMcHaltSlave(Axis:= pAxisRefSlave^, Execute:= FALSE);
			fbMcHome(Axis:= pAxisRefMaster^, Execute:= FALSE);
			fbMcHomingSlave(Axis:= pAxisRefSlave^, Execute:= FALSE);
			fbMcMoveAbs(Axis:= pAxisRefMaster^, Execute:= FALSE);
			fbMcMoveAbsSlave(Axis:= pAxisRefSlave^, Execute:= FALSE);
			fbMcPower(Axis:= pAxisRefMaster^, Enable:= FALSE);
			fbMcPower(Axis:= pAxisRefSlave^, Enable:= FALSE);
			nStateA_Init := 80;
		END_IF
	
	90:	//Error
		//Wenn Antriebe aktiv, dann stoppen
		IF pAxisRefMaster^.Status.Moving OR pAxisRefSlave^.Status.Moving THEN
			nStateA_Init := 91;
		ELSE
			nStateA_Init := 92;
		END_IF

END_CASE

IF nStateA_Init = 91 THEN
		fbMcHalt(Axis:= pAxisRefMaster^ , Execute:= TRUE);
		fbMcHaltSlave(Axis:= pAxisRefSlave^, Execute:= TRUE);
		IF NOT (fbMcHalt.Busy OR fbMcHaltSlave.Busy) THEN
			nStateA_Init := 92;	
		END_IF
ELSIF nStateA_Init = 92 THEN
		fbMcHome(Axis:= pAxisRefMaster^, Execute:= FALSE);
		fbMcHomingSlave(Axis:= pAxisRefSlave^, Execute:= FALSE);
		fbMcMoveAbs(Axis:= pAxisRefMaster^, Execute:= FALSE);
		fbMcMoveAbsSlave(Axis:= pAxisRefSlave^, Execute:= FALSE);
		fbMcPower(Axis:= pAxisRefMaster^, Enable:= FALSE);
		fbMcPower(Axis:= pAxisRefSlave^, Enable:= FALSE);
		fbMcHalt(Axis:= pAxisRefMaster^ , Execute:= FALSE);
		fbMcHaltSlave(Axis:= pAxisRefSlave^, Execute:= FALSE);
		bError := TRUE;
		nStateA_Init := 99;	
END_IF
END_ACTION

ACTION A_PowerOn:
//Nur zum Wiedereinschalten der Antriebe nach einem PowerOff
CASE nStateA_PowerOn OF
	0:	//Slave-Achse ausgekoppelt?
		IF pAxisRefSlave^.Status.Coupled THEN
			nStateA_PowerOn := 1;	//weiter zu auskoppln
		ELSE
			nStateA_PowerOn := 2;
		END_IF
		
	1:	//Slave auskoppeln
		stMethResult := M_GearOut();
		IF NOT stMethResult.bBusy THEN
			IF stMethResult.bError THEN
				nErrorId := stMethResult.nErrorId;
				nStateA_PowerOn := 99;
			ELSE
				nStateA_PowerOn := 2;
			END_IF
		END_IF
		
	2:	//Masterachse freigegeben (einschalten)
		IF NOT pAxisRefMaster^.Status.ControlLoopClosed THEN
			fbMcPower(Axis:= pAxisRefMaster^, Enable:= TRUE, Enable_Positive:= TRUE, Enable_Negative:= TRUE, Override:= 100 );
			IF fbMcPower.Error THEN	 //Fehler bei Ausführung
				nErrorId := UDINT_TO_UINT(fbMcPower.ErrorID);
				fbMcPower(Axis:= pAxisRefMaster^, Enable:= FALSE);
				nStateA_PowerOn := 99;
			END_IF
		ELSE
			nStateA_PowerOn := 3;
		END_IF
		
	3:	//Slaveachse freigegeben (einschalten)
		IF NOT pAxisRefSlave^.Status.ControlLoopClosed THEN
			fbMcPower(Axis:= pAxisRefSlave^, Enable:= TRUE, Enable_Positive:= TRUE, Enable_Negative:= TRUE, Override:= 100);
			IF fbMcPower.Error THEN	 //Fehler bei Ausführung
				nErrorId := UDINT_TO_UINT(fbMcPower.ErrorID);
				fbMcPower(Axis:= pAxisRefSlave^, Enable:= FALSE);
				nStateA_PowerOn := 99;
			END_IF
		ELSE
			nStateA_PowerOn := 4;
			IF pAxisRefMaster^.NcToPlc.ActPos > (P_rMaxPos / 1000.0) THEN
				fbMcMoveAbs.Position := P_rMaxPos / 1000.0;
			ELSE
				fbMcMoveAbs.Position := pAxisRefMaster^.NcToPlc.ActPos;
			END_IF
			fbMcMoveAbsSlave.Position := fbMcMoveAbs.Position;
			bFlag1 := TRUE;
			bFlag2 := TRUE;
		END_IF
		
	4:	//Beide Achsen auf aktuellen Wert von Masterachse fahren
		IF bFlag1 XOR fbMcMoveAbs.Busy THEN
			bFlag1 := FALSE;
			fbMcMoveAbs(Axis:= pAxisRefMaster^, Execute:= TRUE, Velocity:= 10.0); 
		END_IF
		
		IF bFlag2 XOR fbMcMoveAbsSlave.Busy THEN
			bFlag2 := FALSE;
			fbMcMoveAbsSlave(Axis:= pAxisRefSlave^, Execute:= TRUE, Velocity:= 10.0);
		END_IF
		
		IF fbMcMoveAbs.Done AND fbMcMoveAbsSlave.Done THEN
			fbMcMoveAbs(Axis:= pAxisRefMaster^, Execute:= FALSE);
			fbMcMoveAbsSlave(Axis:= pAxisRefSlave^, Execute:= FALSE);
			bFlag1 := TRUE;
			bFlag2 := TRUE;
			nStateA_PowerOn := 5;
		END_IF

		IF fbMcMoveAbs.Error	THEN
			nErrorId := UDINT_TO_UINT(fbMcMoveAbs.ErrorID);
			fbMcMoveAbs(Axis:= pAxisRefMaster^, Execute:= FALSE);
			nStateA_PowerOn := 99;
		END_IF
		
		IF fbMcMoveAbsSlave.Error	THEN
			nErrorId := UDINT_TO_UINT(fbMcMoveAbsSlave.ErrorID);
			fbMcMoveAbsSlave(Axis:= pAxisRefSlave^, Execute:= FALSE);
			nStateA_PowerOn := 99;
		END_IF
		
	5:	//Slave an Master ankoppeln
		stMethResult := M_GearIn();
		IF NOT stMethResult.bBusy THEN
			IF stMethResult.bError THEN
				nErrorId := stMethResult.nErrorId;
				nStateA_PowerOn := 99;
			ELSE
				nStateA_PowerOn := 80;
			END_IF
		END_IF		
END_CASE
END_ACTION

ACTION A_Reset:
CASE nStateA_Reset OF
	0:	
		bBusy := TRUE;
		//Slaveachse
		IF pAxisRefSlave^.Status.Error THEN
			IF pAxisRefSlave^.Status.ErrorID = 16#4550 THEN
				nStateA_Reset := 1;
			ELSE
				nStateA_Reset := 2;
			END_IF
		ELSE
			nStateA_Reset := 3;
		END_IF
	
	1:	//Reset Calibration Slaveachse
		fbMcHomingSlave(Axis:= pAxisRefSlave^, Execute:= TRUE, HomingMode:= Tc2_MC2.MC_HomingMode.MC_ResetCalibration);
		IF NOT fbMcHomingSlave.Busy THEN
			fbMcHomingSlave(Axis:= pAxisRefSlave^, Execute:= FALSE);
			nStateA_Reset := 2;
		END_IF
	
	2:	//Reset Slaveachse
		fbMcReset(Axis:= pAxisRefSlave^, Execute:= TRUE);
		IF NOT fbMcReset.Busy THEN
			fbMcReset(Axis:= pAxisRefSlave^, Execute:= FALSE);
			nStateA_Reset := 3;
		END_IF
		
	3:	//Masterachse
		IF pAxisRefMaster^.Status.Error THEN
			IF pAxisRefMaster^.Status.ErrorID = 16#4550 THEN
				nStateA_Reset := 4;
			ELSE
				nStateA_Reset := 5;
			END_IF
		ELSE
			nStateA_Reset := 6;
		END_IF
		
	4:	//Reset Calibration Masterachse
		fbMcHome(Axis:= pAxisRefMaster^, Execute:= TRUE, HomingMode:= Tc2_MC2.MC_HomingMode.MC_ResetCalibration);
		IF NOT fbMcHome.Busy THEN
			fbMcHome(Axis:= pAxisRefMaster^, Execute:= FALSE);
			nStateA_Reset := 5;
		END_IF
	
	5:	//Reset Masterachse
		fbMcReset(Axis:= pAxisRefMaster^, Execute:= TRUE);
		IF NOT fbMcReset.Busy THEN
			fbMcReset(Axis:= pAxisRefMaster^, Execute:= FALSE);
			nStateA_Reset := 6;
		END_IF
		
	6:	//Checken, ob beide Achsen fehlerfrei
		IF pAxisRefMaster^.Status.Error OR pAxisRefSlave^.Status.Error THEN
			nStateA_Reset := 99;
		ELSE
			//Motion-Bausteine zurücksetzen
			fbMcMoveAbs(Axis:= pAxisRefMaster^, Execute:= FALSE);
			fbMcMoveRel(Axis:= pAxisRefMaster^, Execute:= FALSE);
			fbMcHalt(Axis:= pAxisRefMaster^, Execute:= FALSE);
			fbMcHaltSlave(Axis:= pAxisRefSlave^, Execute:= FALSE);
			nStateA_Reset := 80;
			nStateA_Error := 0;
			bError := FALSE;
		END_IF
END_CASE
END_ACTION

ACTION A_Setup:
CASE nStateA_Setup OF
	0:	bSetupWaitForResp := FALSE;
		bContinueSetup := FALSE;
		//Negativen LimitSwitch deaktivieren(notwendig, da nach Referenzpunkt anfahren auf "0" gefahren wird
		fbMcWriteBoolParameter(Axis:= pAxisRefMaster^, Execute:= TRUE, ParameterNumber:= MC_AxisParameter.EnableLimitNeg, Value:= FALSE);
		IF NOT fbMcWriteBoolParameter.Busy THEN
			IF fbMcWriteBoolParameter.Error THEN
				nStateA_Setup := 99;
			ELSE
				bInit := TRUE;	//Start "Init" auf HomePos "0" (HomePos wird in M_Setup(..) gesetzt)
				nStateA_Setup := 1;
			END_IF
			fbMcWriteBoolParameter(Axis:= pAxisRefMaster^, Execute:= FALSE);
		END_IF
		
	1:	//Warten bis "Init" fertig"
		//danach Achsen auf halbe Workplate + 100 fahren
		IF NOT bInit THEN
			IF bStop THEN
				nStateA_Setup := 5;//weiter zu ResetCalib
			ELSE
				fbMcMoveAbs.Position := rWorkplateLength / 2000.0 - 100.0;
				fbMcMoveAbs.Velocity := 40.0;
				fbMcMoveAbs(Axis:= pAxisRefMaster^, Execute:= TRUE);
				nStateA_Setup := 2;			
			END_IF
		END_IF
		
		IF bError THEN
			bSetupError := TRUE;
			nStateA_Setup := 8; //neg. LimitSwitch wieder aktivieren
		END_IF
		
	2:	//Warten bis Move fertig
		IF bStop THEN
			nStateA_Setup := 50; //weiter zu Stop
		ELSE
			fbMcMoveAbs(Axis:= pAxisRefMaster^, Execute:= TRUE);
			IF fbMcMoveAbs.Error THEN
				nStateA_Setup := 99;
			END_IF
	
			IF NOT fbMcMoveAbs.Busy THEN
				fbMcMoveAbs(Axis:= pAxisRefMaster^, Execute:= FALSE);
				nStateA_Setup := 3;
			END_IF
		END_IF
		
	3:	//Slave auskoppeln
		stMethResult := M_GearOut();
		IF NOT stMethResult.bBusy THEN
			IF stMethResult.bError THEN
				nStateA_Setup := 99;
			ELSE
				nStateA_Setup := 4;
			END_IF
		END_IF

	4:	//beide Achsen ausschalten
		fbMcPower(Axis:= pAxisRefMaster^, Enable:= FALSE);
		fbMcPower(Axis:= pAxisRefSlave^, Enable:= FALSE);
		pAxisRefMaster^.ReadStatus();
		pAxisRefSlave^.ReadStatus();
		IF NOT (pAxisRefMaster^.Status.ControlLoopClosed OR pAxisRefSlave^.Status.ControlLoopClosed) THEN
			nStateA_Setup := 5;
		END_IF
		
	5:	//Calibration Master zurücksetzen
		fbMcHome(Axis:= pAxisRefMaster^, Execute:= TRUE, HomingMode:= MC_ResetCalibration);
		fbMcHomingSlave(Axis:= pAxisRefSlave^, Execute:= TRUE, HomingMode:= MC_ResetCalibration);
		
		IF NOT fbMcHome.Busy AND NOT fbMcHome.Busy THEN
			IF fbMcHome.Error OR fbMcHomingSlave.Error THEN
				nStateA_Setup := 99;
			ELSE
				IF bStop THEN
					nStateA_Setup := 80;
				ELSE
					nStateA_Setup := 6;
					bSetupWaitForResp := TRUE;
					bContinueSetup := FALSE;
				END_IF
			END_IF
			fbMcHome(Axis:= pAxisRefMaster^, Execute:= FALSE);
			fbMcHomingSlave(Axis:= pAxisRefSlave^, Execute:= FALSE);
		END_IF
		
	6:	//Warte auf UserResponse
		IF bContinueSetup THEN
			nStateA_Setup := 7;
		ELSIF bStop THEN
			nStateA_Setup := 8;
		END_IF		
		
	7:	//Neue Referenzposition berechnen und in persistente Variable schreiben
		rRefPosMaster := LREAL_TO_REAL(rWorkplateLength - pAxisRefMaster^.NcToPlc.ActPos * 1000.0 - rNullPosDist - rSetupPosDist);
		rRefPosSlave := LREAL_TO_REAL(rWorkplateLength - pAxisRefSlave^.NcToPlc.ActPos * 1000.0 - rNullPosDist - rSetupPosDist);
		bSetupOK := TRUE;
		nStateA_Setup := 8;
		fbSettings.M_WritePersData();
		
	8:	//Negativen Limit-Switch wieder aktivieren
		fbMcWriteBoolParameter(Axis:= pAxisRefMaster^, Execute:= TRUE, ParameterNumber:= MC_AxisParameter.EnableLimitNeg, Value:= TRUE);
		IF NOT fbMcWriteBoolParameter.Busy THEN
			IF fbMcWriteBoolParameter.Error THEN
				nStateA_Setup := 99;
			ELSE
				IF bSetupError THEN
					nStateA_Setup := 99;
				ELSE
					nStateA_Setup := 80;
				END_IF
			END_IF
			fbMcWriteBoolParameter(Axis:= pAxisRefMaster^, Execute:= FALSE);
		END_IF
	
	50:	//Stop Antriebe (noch im gekoppeltem Zustand)
		fbMcHalt(Axis:= pAxisRefMaster^, Execute:= TRUE);
		IF NOT fbMcHalt.Busy THEN
			fbMcHalt(Axis:= pAxisRefMaster^, Execute:= FALSE);
			nStateA_Setup := 51;
		END_IF
		
	51:	//Falls fbMoveAbs noch busy, dann zu ende führen
		IF fbMcMoveAbs.Busy THEN
			fbMcMoveAbs(Axis:= pAxisRefMaster^);
		ELSE
			fbMcMoveAbs(Axis:= pAxisRefMaster^, Execute := FALSE);
			nStateA_Setup := 3;
		END_IF
	
END_CASE
END_ACTION

METHOD FB_init : BOOL
VAR_INPUT
	bInitRetains 	: BOOL; // if TRUE, the retain variables are initialized (warm start / cold start)
	bInCopyCode 	: BOOL;  // if TRUE, the instance afterwards gets moved into the copy code (online change)
	eXYOrientation	: E_XYOrientation;
	pNCAxisRefMaster: POINTER TO AXIS_REF;
	pNCAxisRefSlave : POINTER TO AXIS_REF;
END_VAR
pAxisRefSlave := pNCAxisRefSlave;
END_METHOD

METHOD M_GearIn : ST_MethResult

VAR_INST
	fbMcGearIn				: Tc2_MC2.MC_GearIn;	//Zum Koppeln der Slave-Achse an die Master-Achse
END_VAR
fbMcGearIn(Master:= pAxisRefMaster^, Slave:= pAxisRefSlave^, Execute:= TRUE,
			RatioNumerator:= 1.0, RatioDenominator:= 1, Busy=> M_GearIn.bBusy, Error=> M_GearIn.bError);
IF NOT fbMcGearIn.Busy THEN
	M_GearIn.nErrorId := UDINT_TO_UINT(fbMcGearIn.ErrorID);
	fbMcGearIn(Master:= pAxisRefMaster^, Slave:= pAxisRefSlave^, Execute:= FALSE);
END_IF
END_METHOD

METHOD M_GearOut : ST_MethResult

VAR_INST
	fbMcGearOut	: Tc2_MC2.MC_GearOut;	//Zum Auskoppeln der Slave-Achse von der Master-Achse
END_VAR
fbMcGearOut(Slave:= pAxisRefSlave^, Execute:= TRUE, Busy=> M_GearOut.bBusy, Error=> M_GearOut.bError);
IF NOT fbMcGearOut.Busy THEN
	IF fbMcGearOut.Error THEN
		M_GearOut.nErrorId := UDINT_TO_UINT(fbMcGearOut.ErrorID);	
	END_IF
	fbMcGearOut(Slave:= pAxisRefSlave^, Execute := FALSE);
END_IF
END_METHOD

METHOD M_GetProperty : ERRORID
VAR_INPUT
	eType	: E_HardwarePropType;
END_VAR
VAR_OUTPUT
	nValue 	: DINT;
END_VAR
IF eType = E_HardwarePropType.RefPos2 THEN
	nValue := REAL_TO_DINT(rRefPosSlave);
ELSE
	M_GetProperty := SUPER^.M_GetProperty(eType,nValue=>nValue);
END_IF
END_METHOD

METHOD M_Init : ERRORID
VAR_INPUT
	bReInit : BOOL;
END_VAR
IF bBusy THEN
	M_Init := E_ErrorIdCmd.ERRORID_AxisStillBusy;
ELSE
	THIS^.bReInit := bReInit;
	//Die Action wird von hier aus einmalig ausgeführt damit ein Aufruf schon in diesem Zyklus stattfindet
	rHomePos := rRefPosMaster / 1000.0;
	rHomePosSlave := rRefPosSlave / 1000.0;
	bInit := TRUE;
	A_Init();		
END_IF
END_METHOD

METHOD M_Jog : ERRORID
VAR_INPUT
	bForward	: BOOL;
	bBackward	: BOOL;
	bInching	: BOOL;
	rDistance	: REAL;
	rSpeed		: REAL;
END_VAR
IF NOT pAxisRefSlave^.Status.Coupled THEN
	M_Jog := E_ErrorIdCmd.ERRORID_X2AxisNotCoupled;
ELSE
	M_Jog := SUPER^.M_Jog(bForward:= bForward, bBackward:= bBackward, bInching:= bInching, rDistance:= rDistance, rSpeed:= rSpeed);
END_IF
END_METHOD

METHOD M_MoveAbs : ERRORID
VAR_INPUT
	rPosition 		: REAL;
	rSpeed			: REAL;
	rAcceleration 	: REAL;
	rDeceleration 	: REAL;
END_VAR
IF NOT pAxisRefSlave^.Status.Coupled THEN
	M_MoveAbs := E_ErrorIdCmd.ERRORID_X2AxisNotCoupled;
ELSE
	M_MoveAbs:= SUPER^.M_MoveAbs(rPosition:= rPosition, rSpeed:= rSpeed, rAcceleration:= rAcceleration, rDeceleration:= rDeceleration);
END_IF
END_METHOD

METHOD M_MoveRel : ERRORID
VAR_INPUT
	rDistance		: REAL;
	rSpeed			: REAL;
	rAcceleration 	: REAL;
	rDeceleration 	: REAL;
END_VAR
IF NOT pAxisRefSlave^.Status.Coupled THEN
	M_MoveRel := E_ErrorIdCmd.ERRORID_X2AxisNotCoupled;
ELSE
	M_MoveRel := SUPER^.M_MoveRel(rDistance:= rDistance, rSpeed:= rSpeed, rAcceleration:= rAcceleration, rDeceleration:= rDeceleration);
END_IF
END_METHOD

METHOD M_PowerOff : ERRORID
VAR_INPUT
END_VAR
fbMcPower(Axis:= pAxisRefMaster^, Enable:= FALSE);
fbMcPower(Axis:= pAxisRefSlave^, Enable:= FALSE);
END_METHOD

METHOD M_PowerOn : ERRORID
VAR_INPUT
END_VAR
IF pAxisRefMaster^.Status.Homed AND pAxisRefSlave^.Status.Homed AND NOT P_bBusy THEN
	bPowerOn := TRUE;
END_IF
END_METHOD

METHOD M_SetProperty : ERRORID
VAR_INPUT
	eType	: E_HardwarePropType;
	nValue 	: DINT;
END_VAR
IF eType = E_HardwarePropType.RefPos2 THEN
	rRefPosSlave := DINT_TO_REAL(nValue);
ELSE
	M_SetProperty := SUPER^.M_SetProperty(eType, nValue);
END_IF
END_METHOD

METHOD M_Setup : ERRORID
VAR_INPUT
END_VAR
IF bBusy THEN
	M_Setup := E_ErrorIdCmd.ERRORID_AxisStillBusy;
ELSE
	THIS^.bReInit := TRUE;
	rHomePos := 0;
	rHomePosSlave := 0;
	bSetup := TRUE;
END_IF
END_METHOD

PROPERTY P_bBusy : BOOL
GET
P_bBusy := SUPER^.P_bBusy OR bPowerOn;
END_GET
END_PROPERTY

PROPERTY P_bCoupled : BOOL
GET
P_bCoupled :=  pAxisRefSlave^.Status.Coupled;
END_GET
END_PROPERTY

PROPERTY P_bIsTwinDrive : BOOL
GET
P_bIsTwinDrive := TRUE;
END_GET
END_PROPERTY

PROPERTY P_pAxisRefSlave : POINTER TO AXIS_REF
GET
P_pAxisRefSlave := pAxisRefSlave;
END_GET
END_PROPERTY

END_FUNCTION_BLOCK

// ---- Hardware/XYDrive/FB_XYDrive_Beck.TcPOU
FUNCTION_BLOCK FB_XYDrive_Beck EXTENDS FB_XYDriveNC
VAR_INPUT
END_VAR
VAR_OUTPUT
END_VAR
VAR

	fbMcAbortTrigger		: Tc2_MC2.MC_AbortTrigger;	//falls Latchvorgang erfolglos abgebrochen
	fbMcTouchProbe			: Tc2_MC2.MC_TouchProbe;
	
	
	stTriggerRef			: TRIGGER_REF := (TouchProbe:= E_TouchProbe.TouchProbe1, Edge:= E_SignalEdge.FallingEdge,
											 Mode:= E_TouchProbeMode.TOUCHPROBEMODE_SINGLE);
											 
	rHomePosSlave : REAL;
	
	bHomeSwitchMaster AT %I* : BOOL;
	
END_VAR

pAxisRefMaster^.ReadStatus();
rActPos := LREAL_TO_REAL(LIMIT(-999.0,pAxisRefMaster^.NcToPlc.ActPos,999.0) * 1000.0);
bHomed := pAxisRefMaster^.Status.Homed;

SUPER^();

ACTION A_Capture:
IF nStateA_Capture = 0 THEN 
	fbMcTouchProbe(Axis:= pAxisRefMaster^, TriggerInput:= stTriggerRef, Execute:= TRUE);
	IF NOT fbMcTouchProbe.Busy AND fbMcTouchProbe.Done THEN
		rCapturedPos := LREAL_TO_REAL(fbMcTouchProbe.RecordedPosition * 1000.0);
		bCaptureOk := TRUE;
		fbMcTouchProbe(Axis:= pAxisRefMaster^, TriggerInput:= stTriggerRef, Execute:= FALSE);
		nStateA_Capture := 80;		
	END_IF
END_IF
END_ACTION

ACTION A_Error:
IF nStateA_Error = 0 THEN
	IF nErrorId = 17744 OR nErrorId = 18000 THEN //Schleppabstandüberwachung "Position" bzw Antriebshardware nicht bereit
		nStateA_Error := 1;
	END_IF
END_IF

CASE nStateA_Error OF
	1:	//Achse ausschalten
		fbMcPower(Axis:= pAxisRefMaster^, Enable:= FALSE);
		IF NOT fbMcPower.Busy THEN
			nStateA_Error := 2;
		END_IF		
	
	2:	//Calibration zurücksetzen
		fbMcHome(Axis:= pAxisRefMaster^, Execute:= TRUE, HomingMode:= MC_ResetCalibration);
		IF NOT fbMcHome.Busy THEN
			IF fbMcHome.Error THEN
				nStateA_Error := 99;
			ELSE
				nStateA_Error := 3;
			END_IF
 			fbMcHome(Axis:= pAxisRefMaster^, Execute:= FALSE);
		END_IF
END_CASE
END_ACTION

ACTION A_Init:
CASE nStateA_Init OF
	0:	//DriveAdress der Achse ermitteln (EncoderId wird für TriggerRef benötigt)
		bBusy := TRUE;
		fbMcReadDriveAddress(Axis:= pAxisRefMaster^ ,Execute:= TRUE, DriveAddress=> stDriveAddress);
		IF NOT fbMcReadDriveAddress.Busy THEN
			IF fbMcReadDriveAddress.Error THEN
				nErrorId := UDINT_TO_UINT(fbMcReadDriveAddress.ErrorID);
				nStateA_Init := 99;
			ELSE
				stTriggerRef.EncoderID := stDriveAddress.NcEncoderId;
				nStateA_Init := 1;
			END_IF
			fbMcReadDriveAddress(Axis:= pAxisRefMaster^ ,Execute:= FALSE);
		END_IF

	1:	//Achse im Fehlerzustand?
		IF pAxisRefMaster^.Status.Error OR fbMcReset.Busy  THEN
			fbMcReset(Axis:= pAxisRefMaster^, Execute:= TRUE); 
			IF fbMcReset.Error THEN	//Error beim zurücksetzen
				nErrorId := UDINT_TO_UINT(fbMcReset.ErrorID);
				fbMcReset(Axis:= pAxisRefMaster^, Execute := FALSE);
				nStateA_Init := 99;
			ELSIF fbMcReset.Done THEN
				fbMcReset(Axis:= pAxisRefMaster^, Execute := FALSE);
				nStateA_Init := 2;
			END_IF
		ELSE
			nStateA_Init := 2;
		END_IF
		
	2:	//Achse freigegeben?
		IF NOT pAxisRefMaster^.Status.ControlLoopClosed THEN
			fbMcPower(Axis:= pAxisRefMaster^, Enable:= TRUE, Enable_Positive:= TRUE, Enable_Negative:= TRUE, Override:= 100 );
			IF fbMcPower.Error THEN	 //Error bei Ausführung
				nErrorId := UDINT_TO_UINT(fbMcPower.ErrorID);
				fbMcPower(Axis:= pAxisRefMaster^, Enable:= FALSE);
				nStateA_Init := 99;
			END_IF
		ELSE
			nStateA_Init := 3;
		END_IF

	3:	//TouchProbe abbrechen
		fbMcAbortTrigger(Axis:= pAxisRefMaster^, TriggerInput:= stTriggerRef, Execute:= TRUE);
		IF NOT fbMcAbortTrigger.Busy THEN
			IF fbMcAbortTrigger.Error THEN
				nErrorId := UDINT_TO_UINT(fbMcAbortTrigger.ErrorID);
				nStateA_Init := 99;
			ELSE
				IF NOT bReInit AND pAxisRefMaster^.Status.Homed THEN
					nStateA_Init := 80; //FERTIG!!
				ELSE
					IF bStop THEN
						nStateA_Init := 80;
					ELSE
						nStateA_Init := 4; //Referenzieren	
					END_IF
					
				END_IF
			END_IF
			fbMcAbortTrigger(Axis:= pAxisRefMaster^ ,TriggerInput:= stTriggerRef, Execute:= FALSE);
		END_IF
		
	4:	//In Abhängigkeit von bInitInvers die Suchrichtung für RefNocken setzen
		fbMcWriteBoolParameter(Axis:= pAxisRefMaster^, Execute:= TRUE, ParameterNumber:= MC_AxisParameter.AxisEncoderHomingInvDirCamSearch, Value:= bInvertInitDir);
		IF NOT fbMcWriteBoolParameter.Busy THEN
			IF fbMcWriteBoolParameter.Error THEN
				nStateA_Init := 99;
			ELSE
				IF bStop THEN
					nStateA_Init := 80;
				ELSE
					nStateA_Init := 5;	
				END_IF
				
			END_IF
			fbMcWriteBoolParameter(Axis:= pAxisRefMaster^, Execute:= FALSE);
		END_IF
		
	5:	//In Abhängigkeit von bInitInvers die Suchrichtung für RefSync setzen
		fbMcWriteBoolParameter(Axis:= pAxisRefMaster^, Execute:= TRUE, ParameterNumber:= MC_AxisParameter.AxisEncoderHomingInvDirSyncSearch, Value:= NOT bInvertInitDir);
		IF NOT fbMcWriteBoolParameter.Busy THEN
			IF fbMcWriteBoolParameter.Error THEN
				nStateA_Init := 99;
			ELSE
				IF bStop THEN
					nStateA_Init := 80;
				ELSE
					nStateA_Init := 6;	
				END_IF
				
			END_IF
			fbMcWriteBoolParameter(Axis:= pAxisRefMaster^, Execute:= FALSE);
		END_IF		
	
	6:	//Achse referenzieren
		fbMcHome(Axis:= pAxisRefMaster^,Execute:= TRUE, Position:= rHomePos, HomingMode:= MC_DefaultHoming, bCalibrationCam:= bHomeSwitchMaster);
		IF NOT fbMcHome.Busy THEN
			IF fbMcHome.Error THEN
				nErrorId := UDINT_TO_UINT(fbMcHome.ErrorID);
				fbMcHome(Axis:= pAxisRefMaster^, Execute := FALSE);
				nStateA_Init := 99;
			END_IF
		END_IF
				
		IF fbMcHome.Done  THEN	//Referenzfahrt abgeschlossen
			fbMcHome(Axis:= pAxisRefMaster^, Execute := FALSE);
			nStateA_Init := 7;
		END_IF
		
		IF bStop THEN
			nStateA_Init := 50;
		END_IF
		
	7:	//Achse auf Referenzpunkt fahren
		fbMcMoveAbs(Axis:= pAxisRefMaster^, Execute:= TRUE, Position:= rHomePos, Velocity:= 10.0);
		IF NOT fbMcMoveAbs.Busy THEN
			IF fbMcMoveAbs.Error THEN
				nErrorId := UDINT_TO_UINT(fbMcMoveAbs.ErrorID);
				fbMcMoveAbs(Axis:= pAxisRefMaster^ , Execute:= FALSE);
				nStateA_Init := 99;
			END_IF
		END_IF
		
		IF fbMcMoveAbs.Done THEN
			fbMcMoveAbs(Axis:= pAxisRefMaster^ , Execute:= FALSE);
			bBusy := FALSE;
			nStateA_Init := 80;
		END_IF
		
		IF bStop THEN
			nStateA_Init := 50;
		END_IF
END_CASE

CASE nStateA_Init OF
	50:	//Stop
		fbMcHalt(Axis:= pAxisRefMaster^, Execute:= TRUE);
		IF NOT fbMcHalt.Busy THEN
			nStateA_Init := 51;
			IF fbMcHalt.Error THEN
				nErrorId := UDINT_TO_UINT(fbMcHalt.ErrorID);
				nStateA_Init := 99;
			END_IF
			fbMcHalt(Axis:= pAxisRefMaster^, Execute:= FALSE);
		END_IF
		
	51,99:
		fbMcPower(Axis:= pAxisRefMaster^, Enable:= FALSE);
		fbMcMoveAbs(Axis:= pAxisRefMaster^ , Execute:= FALSE);
		fbMcHome(Axis:= pAxisRefMaster^, Execute:= FALSE);
		IF nStateA_Init = 51 THEN
			nStateA_Init := 80;
		ELSE
			nStateA_Init := 99;	
		END_IF
END_CASE
END_ACTION

ACTION A_Setup:
CASE nStateA_Setup OF
	0:	
		bSetupWaitForResp := FALSE;
		//Negativen LimitSwitch deaktivieren(notwendig, da nach Referenzpunkt anfahren auf "0" gefahren wird
		fbMcWriteBoolParameter(Axis:= pAxisRefMaster^, Execute:= TRUE, ParameterNumber:= MC_AxisParameter.EnableLimitNeg, Value:= FALSE);
		IF NOT fbMcWriteBoolParameter.Busy THEN
			IF fbMcWriteBoolParameter.Error THEN
				nStateA_Setup := 99;
			ELSE
				nStateA_Setup := 1;
			END_IF
			fbMcWriteBoolParameter(Axis:= pAxisRefMaster^, Execute:= FALSE);
		END_IF
	
	1:	//Achsen intitialisieren mit RefPos0
		bInit := TRUE;
		nStateA_Setup := 2;
		
	2:	//Warten bis "Init" fertig"
		//Achsen auf halbe Workplate - 70 fahren (negative Richtung)
		IF NOT bInit THEN
			IF bStop THEN
				nStateA_Setup := 52;
			ELSE
				fbMcMoveAbs.Position := - (rWorkplateLength / 2000.0 - 70.0);
				fbMcMoveAbs.Velocity := 30.0;
				fbMcMoveAbs(Axis:= pAxisRefMaster^, Execute:= TRUE);
				nStateA_Setup := 3;			
			END_IF
		END_IF
		
		IF bError THEN
			nStateA_Setup := 99;
		END_IF
		
	3:	//Warten bis Move fertig
		IF bStop THEN
			nStateA_Setup := 50; //weiter zu Stop
		ELSE
			fbMcMoveAbs(Axis:= pAxisRefMaster^, Execute:= TRUE);
			IF fbMcMoveAbs.Error THEN
				nStateA_Setup := 99;
			END_IF
	
			IF NOT fbMcMoveAbs.Busy THEN
				fbMcMoveAbs(Axis:= pAxisRefMaster^, Execute:= FALSE);
				nStateA_Setup := 4;
			END_IF
		END_IF
		
	4:	//Achse ausschalten
		fbMcPower(Axis:= pAxisRefMaster^, Enable:= FALSE);
		IF NOT fbMcPower.Busy THEN
			nStateA_Setup := 5;
		END_IF
		
		IF bStop THEN
			nStateA_Setup := 50;
		END_IF
		
	5:	//Calibration zurücksetzen
		fbMcHome(Axis:= pAxisRefMaster^, Execute:= TRUE, HomingMode:= MC_ResetCalibration);
		IF NOT fbMcHome.Busy THEN
			IF fbMcHome.Error THEN
				nStateA_Setup := 99;
			ELSE
				nStateA_Setup := 10;
				bSetupWaitForResp := TRUE;
				bContinueSetup := FALSE;
			END_IF
			fbMcHome(Axis:= pAxisRefMaster^, Execute:= FALSE);
			IF bStop THEN
				nStateA_Setup := 80;
			END_IF
		END_IF
		
	10:	//Warte auf UserResponse
		IF bContinueSetup THEN
			nStateA_Setup := 11;
		ELSIF bStop THEN
			nStateA_Setup := 52;
		END_IF
		
	11:	//Negaitiven LimitSwitch aktivieren
		fbMcWriteBoolParameter(Axis:= pAxisRefMaster^, Execute:= TRUE, ParameterNumber:= MC_AxisParameter.EnableLimitNeg, Value:= TRUE);
		IF NOT fbMcWriteBoolParameter.Busy THEN
			IF fbMcWriteBoolParameter.Error THEN
				nStateA_Setup := 99;
			ELSE
				nStateA_Setup := 12;
			END_IF
			fbMcWriteBoolParameter(Axis:= pAxisRefMaster^, Execute:= FALSE);
		END_IF
		
	12:	//Neue Referenzposition berechnen und in persistente Variable schreiben
		rRefPosMaster := LREAL_TO_REAL(ABS(pAxisRefMaster^.NcToPlc.ActPos * 1000.0) - 1000);
		bSetupOK := TRUE;
		nStateA_Setup := 80;
		fbSettings.M_WritePersData();
		
	50:	//Stop
		fbMcHalt(Axis:= pAxisRefMaster^, Execute:= TRUE);
		IF NOT fbMcHalt.Busy THEN
			nStateA_Setup := 51;
			IF fbMcHalt.Error THEN
				nErrorId := UDINT_TO_UINT(fbMcHalt.ErrorID);
				nStateA_Setup := 99;
			END_IF
			fbMcHalt(Axis:= pAxisRefMaster^, Execute:= FALSE);
		END_IF
		
	51:	//Falls fbMoveAbs noch busy, dann zu ende führen
		IF fbMcMoveAbs.Busy THEN
			fbMcMoveAbs(Axis:= pAxisRefMaster^);
		ELSE
			fbMcMoveAbs(Axis:= pAxisRefMaster^, Execute := FALSE);
			nStateA_Setup := 52;
		END_IF	
		
	52:	//Antriebe aus und ResetCalibration
		fbMcPower(Axis:= pAxisRefMaster^, Enable:= FALSE);
		fbMcMoveAbs(Axis:= pAxisRefMaster^ , Execute:= FALSE);
		fbMcHome(Axis:= pAxisRefMaster^, Execute:= TRUE, HomingMode:= MC_ResetCalibration);
		IF NOT fbMcHome.Busy THEN
			IF fbMcHome.Error THEN
				nStateA_Setup := 99;
			ELSE
				nStateA_Setup := 53;
			END_IF
			fbMcHome(Axis:= pAxisRefMaster^, Execute:= FALSE);
		END_IF

	53:	//negativen LimitSwitch wieder aktivieren		
		fbMcWriteBoolParameter(Axis:= pAxisRefMaster^, Execute:= TRUE, ParameterNumber:= MC_AxisParameter.EnableLimitNeg, Value:= TRUE);
		IF NOT fbMcWriteBoolParameter.Busy THEN
			IF fbMcWriteBoolParameter.Error THEN
				nStateA_Setup := 99;
			ELSE
				nStateA_Setup := 80;
			END_IF
			fbMcWriteBoolParameter(Axis:= pAxisRefMaster^, Execute:= FALSE);
		END_IF	
END_CASE
END_ACTION

ACTION A_StopCapture:
IF nStateA_StopCapture = 0 THEN
	fbMcAbortTrigger(Axis:= pAxisRefMaster^, TriggerInput:= stTriggerRef, Execute:= TRUE);
	IF NOT fbMcAbortTrigger.Busy THEN
		fbMcAbortTrigger(Axis:= pAxisRefMaster^, TriggerInput:= stTriggerRef, Execute:= FALSE);
		fbMcTouchProbe(Axis:= pAxisRefMaster^, TriggerInput:= stTriggerRef, Execute:= FALSE);
		bCaptureStopped := TRUE;
		nStateA_StopCapture := 80;
	END_IF
END_IF
END_ACTION

ACTION A_WriteAxisParameter:
IF nStateA_WriteAxisParamter = 0 THEN
	//feststellen, welcher Parameter als nächstes geschrieben werden muss
	IF nStateWriteLimitNegative = 1 THEN
		nStateWriteLimitNegative := 2;
	ELSIF nStateWriteLimitPositive = 1 THEN
		nStateWriteLimitPositive := 2;
	ELSIF nStateWriteNCIFastSpeed = 1 THEN
		nStateWriteNCIFastSpeed := 2;
	ELSE
		nStateWriteLimitNegative := 1;
		nStateWriteLimitPositive := 1;
		nStateWriteNCIFastSpeed := 1;
		nStateA_WriteAxisParamter := 80;
		RETURN;
	END_IF
	
	IF nStateWriteLimitNegative = 2 THEN
		fbMcWriteParameter.ParameterNumber := MC_AxisParameter.SWLimitNeg;
		fbMcWriteParameter.Value := P_rMinPos / 1000.0;
		nStateA_WriteAxisParamter := 1;
	END_IF
	
	IF nStateWriteLimitPositive = 2 THEN
		fbMcWriteParameter.ParameterNumber := MC_AxisParameter.SWLimitPos;
		fbMcWriteParameter.Value := P_rMaxPos / 1000.0;
		nStateA_WriteAxisParamter := 1;
	END_IF

	IF nStateWriteNCIFastSpeed = 2 THEN
		fbMcWriteParameter.ParameterNumber := MC_AxisParameter.AxisRapidTraverseVelocity;
		fbMcWriteParameter.Value := rMaxSpeed / 1000.0;
		nStateA_WriteAxisParamter := 1;
	END_IF
	
END_IF

IF nStateA_WriteAxisParamter = 1 THEN
	fbMcWriteParameter(Axis:= pAxisRefMaster^, Execute:= TRUE);
	//Hier kann es passieren, dass der Fehler "1793" auftritt. Das passiert manchmal beim Start der SPS
	//In diesem Falle, sollte es solange probiert werden, bis dieser nicht mehr auftritt
	IF NOT fbMcWriteParameter.Busy THEN
		IF fbMcWriteParameter.Error THEN
			IF fbMcWriteParameter.ErrorID <> 1793 THEN
				nStateA_WriteAxisParamter := 99;
			END_IF
		ELSE
			CASE fbMcWriteParameter.ParameterNumber OF
				MC_AxisParameter.SWLimitNeg:
					nStateWriteLimitNegative := 3;
				MC_AxisParameter.SWLimitPos:
					nStateWriteLimitPositive := 3;
				MC_AxisParameter.AxisRapidTraverseVelocity:
					nStateWriteNCIFastSpeed := 3;
			END_CASE
			nStateA_WriteAxisParamter := 0;
		END_IF
		fbMcWriteParameter(Axis:= pAxisRefMaster^, Execute:= FALSE);
	END_IF	
END_IF
END_ACTION

METHOD FB_init : BOOL
VAR_INPUT
	bInitRetains 	: BOOL; // if TRUE, the retain variables are initialized (warm start / cold start)
	bInCopyCode 	: BOOL;  // if TRUE, the instance afterwards gets moved into the copy code (online change)
	eXYOrientation	: E_XYOrientation;
	pNCAxisRefMaster: POINTER TO AXIS_REF;
END_VAR
pAxisRefMaster := pNCAxisRefMaster;
END_METHOD

METHOD M_Capture : ERRORID
VAR_INPUT
END_VAR
bCapture := TRUE;
bCaptureOk := FALSE;
bCaptureStopped := FALSE;
A_Capture();
END_METHOD

METHOD M_Init : ERRORID
VAR_INPUT
	bReInit : BOOL;
END_VAR
IF bBusy THEN
	M_Init := E_ErrorIdCmd.ERRORID_AxisStillBusy;
ELSE
	THIS^.bReInit := bReInit;
	//Die Action wird von hier aus einmalig ausgeführt damit ein Aufruf schon in diesem Zyklus stattfindet
	rHomePos := rRefPosMaster / 1000.0;
	bInit := TRUE;
	A_Init();		
END_IF
END_METHOD

METHOD M_SetProperty : ERRORID
VAR_INPUT
	eType	: E_HardwarePropType;
	nValue 	: DINT;
END_VAR
CASE eType OF
	E_HardwarePropType.RefPos1:
		rRefPosMaster := DINT_TO_REAL(nValue);
	E_HardwarePropType.MinPos:
		M_SetProperty := E_ErrorIdCmd.ERRORID_OnlyReadHwProp;
	E_HardwarePropType.MaxPos:
		M_SetProperty := E_ErrorIdCmd.ERRORID_OnlyReadHwProp;
	E_HardwarePropType.LimitMargeNeg:
		rLimitMargeNeg := DINT_TO_REAL(nValue);
		bWriteAxisParameter := TRUE;
	E_HardwarePropType.LimitMargePos:
		rLimitMargePos := DINT_TO_REAL(nValue);
		bWriteAxisParameter := TRUE;
	E_HardwarePropType.MaxSpeed:
		rMaxSpeed := DINT_TO_REAL(nValue);
		bWriteAxisParameter := TRUE;
	E_HardwarePropType.WorkplateDim:
		rWorkplateLength := DINT_TO_REAL(nValue);
		bWriteAxisParameter := TRUE;
	E_HardwarePropType.NullPosDist:
		rNullPosDist := DINT_TO_REAL(nValue);
		bWriteAxisParameter := TRUE;
	E_HardwarePropType.MaxPosDist:
		rMaxPosDist := DINT_TO_REAL(nValue);
		bWriteAxisParameter := TRUE;
	E_HardwarePropType.SetupPosDist:
		rSetupPosDist := DINT_TO_REAL(nValue);
	E_HardwarePropType.InvertInitDir:
		bInvertInitDir := DINT_TO_BOOL(nValue);
ELSE
	M_SetProperty := E_ErrorIdCmd.ERRORID_InvalidHwProperty;	
END_CASE
END_METHOD

END_FUNCTION_BLOCK

// ---- Hardware/XYDrive/FB_XYDriveNC.TcPOU
FUNCTION_BLOCK FB_XYDriveNC EXTENDS FB_XYDriveBase
VAR_INPUT
END_VAR
VAR_OUTPUT
END_VAR
VAR
	fbMcWriteBoolParameter	: Tc2_MC2.MC_WriteBoolParameter;
	fbMcWriteParameter		: Tc2_MC2.MC_WriteParameter;
	fbMcReset				: Tc2_Mc2.MC_Reset;
	fbMcPower				: Tc2_Mc2.MC_Power;
	fbMcJog					: Tc2_MC2.MC_Jog;
	fbMcHome				: Tc2_MC2.MC_Home;										 
	fbMcMoveAbs				: Tc2_MC2.MC_MoveAbsolute;		
	fbMcMoveRel				: Tc2_MC2.MC_MoveRelative;									 
	fbMcHalt				: Tc2_MC2.MC_Halt;
	
	stDriveAddress			: Tc2_MC2.ST_DriveAddress;	//für CoE-Zugriff
	fbMcReadDriveAddress	: MC_ReadDriveAddress;
	pAxisRefMaster	: POINTER TO Tc2_MC2.AXIS_REF;
END_VAR

SUPER^();
IF NOT bBusy THEN
	IF pAxisRefMaster^.Status.Error THEN
		bError := TRUE;
	END_IF
END_IF

ACTION A_Jog:
//für den Fall, dass der aktuelle Mode inkrementell ist, dann muss für Stop McHalt aufgerufen werden
IF nStateA_Jog = 70 OR bStop THEN
	IF fbMcJog.Mode = E_JogMode.MC_JOGMODE_INCHING THEN
		fbMcHalt(Axis:= pAxisRefMaster^, Execute:= TRUE);
		IF NOT fbMcHalt.Busy THEN
			nStateA_Jog := 80;
			IF fbMcHalt.Error THEN
				nErrorId := UDINT_TO_UINT(fbMcHalt.ErrorID);
				nStateA_Jog := 99;
			END_IF
			fbMcHalt(Axis:= pAxisRefMaster^, Execute:= FALSE);
		END_IF
	END_IF
	fbMcJog(Axis:= pAxisRefMaster^, JogForward := FALSE, JogBackwards := FALSE);
ELSE
	fbMcJog(Axis:= pAxisRefMaster^, JogForward := bJogForward, JogBackwards := bJogBackward);	
END_IF

CASE nStateA_Jog OF
	0:
		bBusy := TRUE;
		IF bJogInching THEN
			nStateA_Jog := 1;
		ELSE
			tmrJog(IN:= TRUE, PT:= T#500MS);
			nStateA_Jog := 2;
		END_IF
		
	2:	//Timer abfragen
		tmrJog();
		IF tmrJog.Q THEN
			fbMcJog(Axis:= pAxisRefMaster^, JogForward:= FALSE, JogBackwards:= FALSE);
		END_IF
END_CASE

IF NOT (fbMcJog.Busy OR fbMcHalt.Busy) THEN
	fbMcJog(Axis:= pAxisRefMaster^, JogForward:= FALSE, JogBackwards:= FALSE);
	tmrJog(IN:=FALSE);
	IF fbMcJog.Error THEN
		nStateA_Jog := 99;
	ELSE
		IF nStateA_Jog = 70 THEN
			IF NOT (bJogForward OR bJogBackward) THEN
				nStateA_Jog := 80;
			ELSE
				nStateA_Jog := 0;
			END_IF
		ELSE
			nStateA_Jog := 80;	
		END_IF
	END_IF
END_IF
END_ACTION

ACTION A_MoveAbs:
IF nStateMoveAbs = 0 THEN
		bBusy := TRUE;
		IF bStop THEN
			nStateMoveAbs := 70;
		ELSE
			fbMcMoveAbs(Axis:= pAxisRefMaster^, Execute:= TRUE);
			IF NOT fbMcMoveAbs.Busy THEN
				IF fbMcMoveAbs.Error THEN
					nErrorId := UDINT_TO_UINT(fbMcMoveAbs.ErrorID);
					nStateMoveAbs := 99;
				ELSE
					nStateMoveAbs := 80;
				END_IF
				fbMcMoveAbs(Axis:= pAxisRefMaster^, Execute:= FALSE);
			END_IF	
		END_IF
END_IF	

IF nStateMoveAbs = 70 THEN
	fbMcHalt(Axis:= pAxisRefMaster^, Execute:= TRUE);
	IF NOT fbMcHalt.Busy THEN
		nStateMoveAbs := 71;
		IF fbMcHalt.Error THEN
			nErrorId := UDINT_TO_UINT(fbMcHalt.ErrorID);
			nStateMoveAbs := 99;
		END_IF
		fbMcHalt(Axis:= pAxisRefMaster^, Execute:= FALSE);
	END_IF
ELSIF nStateMoveAbs = 71 THEN	//MoveBaustein zu Ende führen
	IF fbMcMoveAbs.Busy THEN
		fbMcMoveAbs(Axis:= pAxisRefMaster^);
	ELSE
		fbMcMoveAbs(Axis:= pAxisRefMaster^, Execute:= FALSE);
		nStateMoveAbs := 80;
	END_IF
END_IF
END_ACTION

ACTION A_MoveRel:
IF nStateMoveRel = 0 THEN
	bBusy := TRUE;
	IF bStop THEN
		nStateMoveRel := 70;
	ELSE
		fbMcMoveRel(Axis:= pAxisRefMaster^, Execute:= TRUE);
		IF NOT fbMcMoveRel.Busy THEN
			IF fbMcMoveRel.Error THEN
				nErrorId := UDINT_TO_UINT(fbMcMoveRel.ErrorID);
				nStateMoveRel := 99;
			ELSE
				nStateMoveRel := 80;	
			END_IF
			fbMcMoveRel(Axis:= pAxisRefMaster^, Execute:= FALSE);
		END_IF		
	END_IF
END_IF

IF nStateMoveRel = 70 THEN
	fbMcHalt(Axis:= pAxisRefMaster^, Execute:= TRUE);
	IF NOT fbMcHalt.Busy THEN
		nStateMoveRel := 71;
		IF fbMcHalt.Error THEN
			nErrorId := UDINT_TO_UINT(fbMcHalt.ErrorID);
			nStateMoveRel := 99;
		END_IF
		fbMcHalt(Axis:= pAxisRefMaster^, Execute:= FALSE);
	END_IF
ELSIF nStateMoveRel = 71 THEN
	IF fbMcMoveRel.Busy THEN
		fbMcMoveRel(Axis:= pAxisRefMaster^);
	ELSE
		fbMcMoveRel(Axis:= pAxisRefMaster^, Execute:= FALSE);
		nStateMoveRel := 80;
	END_IF
END_IF
END_ACTION

ACTION A_Reset:
CASE nStateA_Reset OF
	0:	
		bBusy := TRUE;
		IF pAxisRefMaster^.Status.Error THEN
			IF pAxisRefMaster^.Status.ErrorID = 16#4550 THEN //Schleppabstand
				nStateA_Reset := 1;
			ELSE
				nStateA_Reset := 2;
			END_IF
		ELSE
			nStateA_Reset := 3;
		END_IF
	
	1:	//Reset Calibration
		fbMcHome(Axis:= pAxisRefMaster^, Execute:= TRUE, HomingMode:= Tc2_MC2.MC_HomingMode.MC_ResetCalibration);
		IF NOT fbMcHome.Busy THEN
			fbMcHome(Axis:= pAxisRefMaster^, Execute:= FALSE);
			nStateA_Reset := 2;
		END_IF
	
	2:	//Reset Achse
		fbMcReset(Axis:= pAxisRefMaster^, Execute:= TRUE);
		IF NOT fbMcReset.Busy THEN
			fbMcReset(Axis:= pAxisRefMaster^, Execute:= FALSE);
			nStateA_Reset := 3;
		END_IF
		
	3:	//Checken, ob Achse fehlerfrei
		IF pAxisRefMaster^.Status.Error THEN
			nStateA_Reset := 99;
		ELSE
			//Motion-Bausteine zurücksetzen
			fbMcMoveAbs(Axis:= pAxisRefMaster^, Execute:= FALSE);
			fbMcMoveRel(Axis:= pAxisRefMaster^, Execute:= FALSE);
			fbMcHalt(Axis:= pAxisRefMaster^, Execute:= FALSE);
			nStateA_Reset := 80;
			nStateA_Error := 0;
			bError := FALSE;
		END_IF
END_CASE
END_ACTION

METHOD FB_init : BOOL
VAR_INPUT
	bInitRetains 	: BOOL; // if TRUE, the retain variables are initialized (warm start / cold start)
	bInCopyCode 	: BOOL;  // if TRUE, the instance afterwards gets moved into the copy code (online change)
	eXYOrientation	: E_XYOrientation;
END_VAR
nStateWriteLimitNegative := 1;
nStateWriteLimitPositive := 1;
nStateWriteNCIFastSpeed := 1;
bWriteAxisParameter := TRUE;
END_METHOD

METHOD M_Jog : ERRORID
VAR_INPUT
	bForward	: BOOL;
	bBackward	: BOOL;
	bInching	: BOOL;
	rDistance	: REAL;
	rSpeed		: REAL;		
END_VAR
bJogForward := bForward;
bJogBackward := bBackward;
fbMcJog.Position := rDistance / 1000.0;
fbMcJog.Velocity := rSpeed / 1000.0;

//Ein Richtungswechsel bzw. Modewechsel sollte immer erst einen Stop ausführen, falls Jog noch aktiv ist.
IF bJog THEN
	IF bForward <> bJogForward OR bBackward <> bJogBackward OR bInching <> bJogInching THEN
		//Stoppen und falls kein Stop angefordert, dann neu mit neuen Paramtern ausführen
		//für diesen Fall müssen die Parameter zwischengespeichert werden?
		nStateA_Jog := 70;
		A_Jog();
	ELSE
		//continuierliches Joggen:
		//Timer zurücksetzen und nStateA_Jog auf "0" setzen
		//inkrementelles Joggen:
		//das letzte Increment sollte erst abgearbeitet sein
		IF bInching THEN
			fbMcJog.Mode := Tc2_MC2.E_JogMode.MC_JOGMODE_INCHING;
		ELSE
			fbMcJog.Mode := Tc2_MC2.E_JogMode.MC_JOGMODE_CONTINOUS;
		END_IF		
		tmrJog(IN:=FALSE);
		nStateA_Jog := 0;
		A_Jog();
	END_IF
ELSE
	IF bBusy THEN
		M_Jog := E_ErrorIdCmd.ERRORID_AxisStillBusy;
	ELSE
		bJog := TRUE;
		IF bInching THEN
			fbMcJog.Mode := Tc2_MC2.E_JogMode.MC_JOGMODE_INCHING;
			bJogInching := TRUE;
		ELSE
			fbMcJog.Mode := Tc2_MC2.E_JogMode.MC_JOGMODE_CONTINOUS;
			bJogInching := FALSE;
		END_IF		
		A_Jog();
	END_IF
END_IF
END_METHOD

METHOD M_MoveAbs : ERRORID
VAR_INPUT
	rPosition 		: REAL;
	rSpeed			: REAL;
	rAcceleration 	: REAL;
	rDeceleration 	: REAL;
END_VAR
IF bBusy THEN
	M_MoveAbs := E_ErrorIdCmd.ERRORID_AxisStillBusy;
ELSE
	fbMcMoveAbs.Position := rPosition / 1000.0;
	
	IF rSpeed < 0 OR rSpeed > rMaxSpeed THEN
		fbMcMoveAbs.Velocity := rMaxSpeed / 1000.0;	
	ELSE
		fbMcMoveAbs.Velocity := rSpeed / 1000.0;
	END_IF
	
	IF rAcceleration > 0 THEN
		fbMcMoveAbs.Acceleration := rAcceleration / 1000.0;
	END_IF
	
	IF rDeceleration > 0 THEN
		fbMcMoveAbs.Deceleration := rDeceleration / 1000.0;
	END_IF
	bMoveAbs := TRUE;
	A_MoveAbs();
END_IF
END_METHOD

METHOD M_MoveRel : ERRORID
VAR_INPUT
	rDistance		: REAL;
	rSpeed			: REAL;
	rAcceleration 	: REAL;
	rDeceleration 	: REAL;	
END_VAR
IF bBusy THEN
	M_MoveRel := E_ErrorIdCmd.ERRORID_AxisStillBusy;
ELSE
	fbMcMoveRel.Distance := rDistance / 1000.0;
	
	IF rSpeed < 0 THEN
		fbMcMoveRel.Velocity := rMaxSpeed / 1000.0;	
	ELSE
		fbMcMoveRel.Velocity := rSpeed / 1000.0;
	END_IF
	
	IF rAcceleration > 0 THEN
		fbMcMoveRel.Acceleration := rAcceleration / 1000.0;
	END_IF
	
	IF rDeceleration > 0 THEN
		fbMcMoveRel.Deceleration := rDeceleration / 1000.0;
	END_IF
	bMoveRel := TRUE;
	A_MoveRel();
END_IF
END_METHOD

METHOD M_PowerOff : ERRORID
VAR_INPUT
END_VAR
fbMcPower(Axis:= pAxisRefMaster^, Enable:= FALSE, Enable_Positive:= TRUE, Enable_Negative:= TRUE, Override:= 100);
END_METHOD

METHOD M_PowerOn : ERRORID
VAR_INPUT
END_VAR
IF pAxisRefMaster^.Status.Homed THEN
	fbMcPower(Axis:= pAxisRefMaster^, Enable:= TRUE, Enable_Positive:= TRUE, Enable_Negative:= TRUE, Override:= 100 );
	IF pAxisRefMaster^.Status.Error THEN
		nErrorId := UDINT_TO_UINT(pAxisRefMaster^.Status.ErrorID);
		bError := TRUE;
	END_IF
END_IF
END_METHOD

PROPERTY P_bCoupled : BOOL
GET
//Wird nur zur Kopplung YY bei 2-Ebenen verwendet
P_bCoupled := pAxisRefMaster^.Status.Coupled;
END_GET
END_PROPERTY

PROPERTY P_bIsMoving : BOOL
GET
pAxisRefMaster^.ReadStatus();
P_bIsMoving :=  pAxisRefMaster^.Status.Moving;
END_GET
END_PROPERTY

PROPERTY P_pAxisRef : POINTER TO AXIS_REF
GET
P_pAxisRef := pAxisRefMaster;
END_GET
END_PROPERTY

END_FUNCTION_BLOCK

// ---- GCode/FB_ClearGroup.TcPOU
FUNCTION_BLOCK FB_ClearGroup
VAR_INPUT
	bExecute	: BOOL;
	bReGearInSlave : BOOL;
END_VAR
VAR_OUTPUT
	bBusy		: BOOL;
	bError		: BOOL;
	nErrorId	: ERRORID;	
END_VAR
VAR_IN_OUT
	stGCodeRef : ST_GCodeRef;
END_VAR
VAR
	nState				: USINT;
	fbCfgReconfigGroup	: Tc2_NCI.CfgReconfigGroup;
	fbMcGearIn			: Tc2_MC2.MC_GearIn;
	fbMcGearOut			: Tc2_MC2.MC_GearOut;
	pNciToPlc 			: POINTER TO NCTOPLC_NCICHANNEL_REF;
	pXDrive				: POINTER TO FB_XYDriveBase;
	pYDrive				: POINTER TO FB_XYDriveBase;
	pTwinDrive			: POINTER TO FB_XYDrive_Beck_Twin;;
END_VAR

IF bExecute THEN
	IF nState = 0 THEN	//X-Slave-Achse gekoppelt?
		pNciToPlc := ADR(stGCodeRef.sNciToPlc);
		IF stGCodeRef.pHead = 0 THEN //GCode wurde noch nicht benutzt und entsprechend braucht auch keine Gruppe gelöscht werden
			RETURN;	
		END_IF
		pXDrive := stGCodeRef.pHead^.P_pXDrive;
		pYDrive := stGCodeRef.pHead^.P_pYDrive;
		bBusy := TRUE;
		IF pXDrive^.P_bIsTwinDrive AND_THEN pXDrive^.P_bCoupled THEN
			pTwinDrive := pXDrive;
			nState := 1;
		ELSE
			nState := 2;
		END_IF		
	END_IF
	
	IF nState = 1 THEN	//X-Slave auskopplen
		fbMcGearOut(Slave := pTwinDrive^.P_pAxisRefSlave^, Execute:= TRUE);
		IF NOT fbMcGearOut.Busy THEN
			IF fbMcGearOut.Error THEN
				nErrorId := UDINT_TO_UINT(fbMcGearOut.ErrorID);
				nState := 99;
			ELSE
				nState := 2;
			END_IF
			fbMcGearOut(Slave := pTwinDrive^.P_pAxisRefSlave^, Execute:= FALSE);
		END_IF
	END_IF	

	IF nState = 2 THEN
		fbCfgReconfigGroup(bExecute:= TRUE, nGroupId:= ItpGetGroupId(pNciToPlc^));
		IF NOT fbCfgReconfigGroup.bBusy THEN
			IF fbCfgReconfigGroup.bErr THEN
				nErrorId := UDINT_TO_UINT(fbCfgReconfigGroup.nErrId);
				nState := 99;
			ELSE
				IF bReGearInSlave AND pXDrive^.P_bIsTwinDrive THEN
					pTwinDrive := pXDrive;
					nState := 3;
				ELSE
					bBusy := FALSE;
					nState := 80;
				END_IF
			END_IF
			fbCfgReconfigGroup(bExecute:= FALSE);
		END_IF		
	END_IF	

	IF nState = 3 THEN	//X-Slave einkopplen
		fbMcGearIn(Master:= pTwinDrive^.P_pAxisRef^, Slave:= pTwinDrive^.P_pAxisRefSlave^, Execute:= TRUE, RatioNumerator:= 1.0);
		IF NOT fbMcGearIn.Busy THEN
			IF fbMcGearIn.Error THEN
				nErrorId := UDINT_TO_UINT(fbMcGearIn.ErrorID);
				nState := 99;
			ELSE
				bBusy := FALSE;
				nState := 80;
			END_IF
			fbMcGearIn(Master:= pTwinDrive^.P_pAxisRef^, Slave:= pTwinDrive^.P_pAxisRefSlave^, Execute:= FALSE);
		END_IF		
	END_IF
	
	IF nState = 99 THEN
		bError := TRUE;
		bBusy := FALSE;	
	END_IF	

ELSE
	bError := FALSE;
	nErrorId := 0;
	nState := 0;	
END_IF

END_FUNCTION_BLOCK

// ---- GCode/FB_HskMFunc.TcPOU
FUNCTION_BLOCK FB_HskMFunc
VAR_INPUT
	bStop 		: BOOL;	//hat Vorrang vor bPause und bContinue
	bPause		: BOOL;	//nicht alle M-Funktionen lassen sich pausieren, hat Vorrang vor bContinue
	bContinue	: BOOL; //falls in Pause, dann Fortsetzung
END_VAR
VAR_OUTPUT
	bBusy				: BOOL;
	bError				: BOOL;
	nErrorId			: ERRORID;
	bCanceled			: BOOL;
	bIsInPause			: BOOL;
END_VAR
VAR_IN_OUT
	stGCodeRef			: ST_GCodeRef;
	pXDrive				: POINTER TO FB_XYDriveBase;
	pYDrive				: POINTER TO FB_XYDriveBase;	
END_VAR
VAR
	nStateAction		: USINT;
	nMFuncNumber		: UINT;
	bMFuncRequest		: BOOL;
	bMFuncConfirm		: BOOL;
	stActionData		: ST_ActionData;
	alrRParam			: ARRAY[1..cMaxRParams] OF LREAL;
	ePrintParamType		: E_PrintParamType;
	nPrintParamNumerator: USINT;
	nPrintParamValue	: DINT;
	stMethResult		: ST_MethResult;
	
	rTrig				: R_TRIG;
	fbItpReadRParams	: Tc2_NCI.ItpReadRParamsEx;
	fbItpReadRParamsHdr	: Tc2_NCI.ItpReadRParamsEx; //Lesen des Headers
	fbItpWriteRParams	: Tc2_NCI.ItpWriteRParamsEx;
	fbItpWriteZeroShiftEx	: Tc2_NCI.ItpWriteZeroShiftEx;	//Zum Schreiben der Nullpunktverschiebung
	fbItpConfirmHsk 		: Tc2_NCI.ItpConfirmHsk;
	
	fbMcSetPosition		: Tc2_Mc2.MC_SetPosition;
	pNewTool			: POINTER TO FB_GCodeTool;
	pPiezoPip			: POINTER TO FB_PiezoPip;
	pPassivPip			: POINTER TO FB_PassivPip;
	pExtruder			: POINTER TO FB_Extruder;
	pTwinExtruder		: POINTER TO FB_TwinExtruder;
	pTwinPiezoHolder	: POINTER TO FB_TwinPiezoHolder;
	pTarget				: POINTER TO FB_TargetBase;
	pMultiCartHolder	: POINTER TO FB_MultiCartHolder;
	pHybridDispenser	: POINTER TO FB_HybridDispenser;
	pMtp				: POINTER TO FB_Mtp;
	pVialRack			: POINTER TO FB_VialRack;
	pPieceSlot			: POINTER TO FB_PieceSlot;

	stError 			: ST_Error := (POU := E_POU.POU_FB_HskMFunc);
	fbBuildGroup		: FB_BuildGroup();
	fbClearGroup		: FB_ClearGroup();
	
	alrHeaderRParam		: ARRAY[101..125] OF LREAL;
	i					: USINT;
	nCyclCounter		: USINT;
	nToolNr				: USINT;
		
	sSetPositionOptions		: Tc2_Mc2.ST_SetPositionOptions := (ClearPositionLag:= TRUE);
	
	stPos1				: ST_3DPoint;
	stPos2				: ST_3DPoint;
	stCurrentPos		: ST_3DPoint;
	
	tDelay				: TIME;
	nChannel			: USINT;
	timer				: TON;
	
	stMeasToolOldOffset	: ST_3DPoint;
	stMeasToolNewOffset	: ST_3DPoint;
	
	nSequenceNr			: UINT;
	pSequence			: POINTER TO FB_Sequence;
	
	nStateA_MoveBack	: USINT;
	nStateA_MoveFree	: USINT;
	
	//PipPre- und PostSequence
	nTgtNrWS_Wash1 		: UINT;
	nSpecPointNr_Wash1 	: UINT;
	nWashFlow_Wash1		: DINT;
	nWashTime_Wash1		: DINT;
	nTgtNrWS_Wash2 		: UINT;
	nSpecPointNr_Wash2 	: UINT;
	nWashFlow_Wash2		: DINT;
	nWashTime_Wash2		: DINT;
	nTgtNrDryPad_Dry1	: UINT;
	nDryCount_Dry1		: USINT;
	nDryTime_Dry1		: DINT;
	nTgtNrDryPad_Dry2	: UINT;
	nDryCount_Dry2		: USINT;
	nDryTime_Dry2		: DINT;
	nTgtNrSource		: UINT; //Mtp oder VialRack für GetSample
	nGetSampleColSlotNr	: DINT; //Col bei Mtp, SlotNr bei VialRack
	nGetSampleRow		: DINT;
	nGetSampleQuantity	: DINT;
	nGetSampleFlow		: DINT;
	nGetSampleDelay		: DINT;
	nGetSampleAirGap	: DINT;
	nGetSampleDilBypass	: DINT;
	nTgtNrStrob			: UINT;
	nDispenseTest		: DINT;
	
	nTgtNrWS_DispenseWaste1		: UINT;
	nSpecPointNr_DispenseWaste1 : UINT;
	nQuantity_DispenseWaste1	: DINT;
	nFlow_DispenseWaste1		: DINT;
	
	nTgtNrWS_DispenseWaste2		: UINT;
	nSpecPointNr_DispenseWaste2 : UINT;
	nQuantity_DispenseWaste2	: DINT;
	nFlow_DispenseWaste2		: DINT;
	
	//UniDispense
	nUniDispParam1 : DINT;
	nUniDispParam2 : DINT;
	bUnitDispIsContinous : BOOL;
	
END_VAR

VAR CONSTANT
	cMaxRParams : USINT := 27;
END_VAR

bMFuncRequest := ItpIsHskMFunc(stGCodeRef.sNciToPlc);
nMFuncNumber := INT_TO_UINT(ItpGetHskMFunc(stGCodeRef.sNciToPlc));

rTrig(CLK:= bMFuncRequest);

IF rTrig.Q THEN
	fbItpReadRParams(sNciToPlc:= stGCodeRef.sNciToPlc, bExecute:= TRUE, pAddr:= ADR(alrRParam), nIndex:= 1, nCount:= cMaxRParams);
END_IF

fbItpReadRParams(sNciToPlc:= stGCodeRef.sNciToPlc);
IF NOT fbItpReadRParams.bBusy AND fbItpReadRParams.bExecute THEN
	fbItpReadRParams(sNciToPlc:= stGCodeRef.sNciToPlc, bExecute:= FALSE);
END_IF

IF bMFuncRequest OR bMFuncConfirm THEN
	bBusy := TRUE;
END_IF

IF bMFuncRequest AND NOT bMFuncConfirm THEN
	CASE nMFuncNumber OF
		5:	//RParameter Header verarbeiten
			A_AssignHeaderRParams();
			IF nStateAction = 80 THEN
				bMFuncConfirm := TRUE;
				nStateAction := 0;
			ELSIF nStateAction = 81 THEN	//Abbruch durch Interaktion (ZSensor mounted)
				bMFuncConfirm := TRUE;
				nStateAction := 0;
				bCanceled := TRUE;
			ELSIF nStateAction = 99 THEN	//Error
				nStateAction := 0;
				stError.POUAction := E_POUACT.POUACT_A_AssignRParamHeader;
				fbErrorList.M_Add(stError);				
				bError := TRUE;
				bBusy := FALSE;
			END_IF
	
		6:	//Select Tool
			A_SelectTool();
			IF nStateAction >= 80 THEN
				IF nStateAction >= 99 THEN
					stError.POUAction := E_POUACT.POUACT_A_SelectTool;
					fbErrorList.M_Add(stError);					
					bError := TRUE;
				END_IF
				nStateAction := 0;
				bMFuncConfirm := TRUE;
			END_IF
			
		101: //MoveZ home
			A_MoveZHome();
			IF nStateAction >= 80 THEN
				IF nStateAction >= 99 THEN
					stError.POUAction := E_POUACT.POUACT_A_MoveZHome;
					fbErrorList.M_Add(stError);					
					bError := TRUE;
				END_IF
				nStateAction := 0;
				bMFuncConfirm := TRUE;
			END_IF
			
		102: //SetPrintParameter
			A_SetPrintParams();
			IF nStateAction >= 80 THEN
				IF nStateAction >= 99 THEN
					stError.POUAction := E_POUACT.POUACT_A_SetPrintParams;
					fbErrorList.M_Add(stError);					
					bError := TRUE;
				END_IF
				nStateAction := 0;
				bMFuncConfirm := TRUE;
			END_IF

		103: //SwitchPress
			A_SwitchPress();
			IF nStateAction >= 80 THEN
				IF nStateAction >= 99 THEN
					stError.POUAction := E_POUACT.POUACT_A_SwitchPress;
					fbErrorList.M_Add(stError);					
					bError := TRUE;
				END_IF
				nStateAction := 0;
				bMFuncConfirm := TRUE;
			END_IF
			
		110: //MeasureTool
			A_MeasureTool();
			IF nStateAction >= 80 THEN
				IF nStateAction >= 99 THEN
					stError.POUAction := E_POUACT.POUACT_A_MeasureTool;
					fbErrorList.M_Add(stError);					
					bError := TRUE;
				END_IF
				nStateAction := 0;
				bMFuncConfirm := TRUE;
			END_IF
			
		111: //CleanTip
			A_CleanTip();
			IF nStateAction >= 80 THEN
				IF nStateAction >= 99 THEN
					stError.POUAction := E_POUACT.POUACT_A_CleanTip;
					fbErrorList.M_Add(stError);					
					bError := TRUE;
				END_IF
				nStateAction := 0;
				bMFuncConfirm := TRUE;
			END_IF

		114: //Aspirate
			A_Aspirate();
			IF nStateAction >= 80 THEN
				IF nStateAction >= 99 THEN
					stError.POUAction := E_POUACT.POUACT_A_Aspirate;
					fbErrorList.M_Add(stError);
					bError := TRUE;
				END_IF
				nStateAction := 0;
				bMFuncConfirm := TRUE;
			END_IF
			
		115: //Dispense
			A_Dispense();
			IF nStateAction >= 80 THEN
				IF nStateAction >= 99 THEN
					stError.POUAction := E_POUACT.POUACT_A_Dispense;
					fbErrorList.M_Add(stError);					
					bError := TRUE;
				END_IF
				nStateAction := 0;
				bMFuncConfirm := TRUE;
			END_IF

		116: //Extrude
			A_Extrude();
			IF nStateAction >= 80 THEN
				IF nStateAction >= 99 THEN
					stError.POUAction := E_POUACT.POUACT_A_Extrude;
					fbErrorList.M_Add(stError);					
					bError := TRUE;
				END_IF
				nStateAction := 0;
				bMFuncConfirm := TRUE;
			END_IF		

		117: //BasicDispense (Hybrid-Dispenser)
			A_BasicDispense();
			IF nStateAction >= 80 THEN
				IF nStateAction >= 99 THEN
					stError.POUAction := E_POUACT.POUACT_A_BasicDispense;
					fbErrorList.M_Add(stError);				
					bError := TRUE;
				END_IF
				nStateAction := 0;
				bMFuncConfirm := TRUE;
			END_IF		
			
		118: //DispenseDrops
			A_DispenseDrops();
			IF nStateAction >= 80 THEN
				IF nStateAction >= 99 THEN
					stError.POUAction := E_POUACT.POUACT_A_DispensePiezo;
					fbErrorList.M_Add(stError);					
					bError := TRUE;
				END_IF
				nStateAction := 0;
				bMFuncConfirm := TRUE;
			END_IF
			
		119: //WaitForUser
			A_WaitForUser();
			IF nStateAction >= 80 THEN
				IF nStateAction >= 99 THEN
					stError.POUAction := E_POUACT.POUACT_A_WaitForUser;
					fbErrorList.M_Add(stError);					
					bError := TRUE;
				END_IF
				nStateAction := 0;
				bMFuncConfirm := TRUE;
			END_IF		

		121: //Expose
			A_Expose();
			IF nStateAction >= 80 THEN
				IF nStateAction >= 99 THEN
					stError.POUAction := E_POUACT.POUACT_A_Expose;
					fbErrorList.M_Add(stError);					
					bError := TRUE;
				END_IF
				nStateAction := 0;
				bMFuncConfirm := TRUE;
			END_IF		
	
		120: //WaitAtPoint
			A_WaitAtPoint();
			IF nStateAction >= 80 THEN
				IF nStateAction >= 99 THEN
					stError.POUAction := E_POUACT.POUACT_A_WaitAtPoint;
					fbErrorList.M_Add(stError);					
					bError := TRUE;
				END_IF
				nStateAction := 0;
				bMFuncConfirm := TRUE;
			END_IF		
			
		122: //RunSequence
			A_Sequence();
			IF nStateAction >= 80 THEN
				IF nStateAction >= 99 THEN
					stError.POUAction := E_POUACT.POUACT_A_Sequence;
					fbErrorList.M_Add(stError);					
					bError := TRUE;
				END_IF
				nStateAction := 0;
				bMFuncConfirm := TRUE;
			END_IF
			
		123: //DilMoveValve (zu Piezo zugehöriger)
			A_DilMoveValve();
			IF nStateAction >= 80 THEN
				IF nStateAction >= 99 THEN
					stError.POUAction := E_POUACT.POUACT_A_DilMoveValve;
					fbErrorList.M_Add(stError);					
					bError := TRUE;
				END_IF
				nStateAction := 0;
				bMFuncConfirm := TRUE;
			END_IF
			
		124: //PipPreSequence
			A_PipPreSequence();
			IF nStateAction >= 80 THEN
				IF nStateAction >= 99 THEN
					stError.POUAction := E_POUACT.POUACT_A_PipPreSequence;
					fbErrorList.M_Add(stError);					
					bError := TRUE;
				END_IF
				nStateAction := 0;
				bMFuncConfirm := TRUE;
			END_IF
			
		125: //PipPostSequence
			A_PipPostSequence();
			IF nStateAction >= 80 THEN
				IF nStateAction >= 99 THEN
					stError.POUAction := E_POUACT.POUACT_A_PipPostSequence;
					fbErrorList.M_Add(stError);					
					bError := TRUE;
				END_IF
				nStateAction := 0;
				bMFuncConfirm := TRUE;
			END_IF

		126: //StirrCartridge
			A_StirrCartridge();
			IF nStateAction >= 80 THEN
				IF nStateAction >= 99 THEN
					stError.POUAction := E_POUACT.POUACT_A_StirrCartridge;
					fbErrorList.M_Add(stError);					
					bError := TRUE;
				END_IF
				nStateAction := 0;
				bMFuncConfirm := TRUE;
			END_IF
			
		127: //UniDispense
			A_UniDispense();
			IF nStateAction >= 80 THEN
				IF nStateAction >= 99 THEN
					stError.POUAction := E_POUACT.POUACT_A_UniDispense;
					fbErrorList.M_Add(stError);					
					bError := TRUE;
				END_IF
				nStateAction := 0;
				bMFuncConfirm := TRUE;
			END_IF
			
		
	END_CASE
END_IF

IF bMFuncConfirm THEN
	fbItpConfirmHsk(bExecute:= TRUE ,sNciToPlc:= stGCodeRef.sNciToPlc, sPlcToNci:= stGCodeRef.sPlcToNci);
	IF NOT fbItpConfirmHsk.bBusy THEN
		IF fbItpConfirmHsk.bErr THEN
			nErrorId := UDINT_TO_UINT(fbItpConfirmHsk.nErrId);
			bError := TRUE;
		END_IF
		fbItpConfirmHsk(bExecute:= FALSE ,sNciToPlc:= stGCodeRef.sNciToPlc, sPlcToNci:= stGCodeRef.sPlcToNci);
		bMFuncConfirm := FALSE;
		bBusy := FALSE;
	END_IF	
END_IF

ACTION A_Aspirate:
stError.POUState := nStateAction;

CASE nStateAction OF
	0:	
		IF bStop THEN
			nStateAction := 80;
		ELSE
			IF stGCodeRef.pCurrentTool = 0 THEN
				stError.ErrorId := E_ErrorIdGCode.ERRORID_NoSelectedTool;
				nStateAction := 99;
			ELSE
				IF NOT fbItpReadRParams.bBusy THEN
					MEMSET(ADR(stActionData),0,SIZEOF(stActionData));
					stActionData.eAction := E_Action.ACTION_Aspirate;
					stActionData.aParams[1] := LREAL_TO_DINT(alrRParam[1]);
					stActionData.aParams[2] := LREAL_TO_DINT(alrRParam[2]);
					stError.ErrorId := stGCodeRef.pCurrentTool^.M_ExeAction(stActionData);
					IF stError.ErrorId > 0 THEN
						nStateAction := 99;
					ELSE
						nStateAction := 1;
					END_IF
				END_IF
			END_IF
		END_IF
		
	1:	//Aspirate ready?
		IF bStop THEN
			stGCodeRef.pCurrentTool^.M_CancelAction(E_Action.ACTION_Aspirate);
		END_IF
		
		IF NOT stGCodeRef.pCurrentTool^.P_bBusy THEN
			IF stGCodeRef.pCurrentTool^.P_bError THEN
				stError.ErrorId := stGCodeRef.pCurrentTool^.P_nErrorId;
				nStateAction := 99;
			ELSE
				nStateAction := 80;	
			END_IF
		END_IF
END_CASE
END_ACTION

ACTION A_AssignHeaderRParams:
stError.POUState := nStateAction;

CASE nStateAction OF
	0:	//R-Parameter R101 bis R125 auslesen
		//R101 bis R120 Toolnummern
		//R121 bis R125 Dimension des Scaffolds
		fbItpReadRParamsHdr(sNciToPlc:= stGCodeRef.sNciToPlc, bExecute:= TRUE, pAddr:= ADR(alrHeaderRParam),nIndex:= 101, nCount:= 25);
		IF NOT fbItpReadRParamsHdr.bBusy THEN
			IF fbItpReadRParamsHdr.bErr THEN
				stError.ErrorId := UDINT_TO_UINT(fbItpReadRParamsHdr.nErrId);
				nStateAction := 99;
			ELSE
				IF bStop THEN
					nStateAction := 80;
				ELSE
					nStateAction := 1;	
				END_IF
			END_IF
			fbItpReadRParamsHdr(sNciToPlc:= stGCodeRef.sNciToPlc, bExecute:= FALSE);
		END_IF

	1:	//ObjectIds zuordnen
		//Die RParams iterieren
		FOR i := 101 TO 110 BY 1 DO
			//als Erstes den RParameter checken
			//er darf nicht größer sein als max Tools
			nToolNr := LREAL_TO_USINT(alrHeaderRParam[i]); //Die R-Parameter werden in GCode auf "0" gesetzt
			IF nToolNr > GCode.cMaxGCodeTools THEN
				stError.ErrorId := E_ErrorIdGCode.ERRORID_InvalidToolNr;		
				nStateAction := 99;
			ELSIF nToolNr > 0 THEN
				IF stGCodeRef.aToolTable[nToolNr].pMzTool > 0 THEN
					IF NOT stGCodeRef.aToolTable[nToolNr].pMzTool^.P_bIsInit THEN
						stError.ObjectId := stGCodeRef.aToolTable[i].pMzTool^.P_nObjectID;
						stError.ErrorId := E_ErrorIdCmd.ERRORID_DeviceNotInitialized;
						nStateAction := 99;
						EXIT;
					END_IF
				ELSE
					stError.ErrorId := E_ErrorIdGCode.ERRORID_InvalidToolNr;		
					nStateAction := 99;
				END_IF
				stGCodeRef.aToolTable[nToolNr].bIsUsed := TRUE; //Dieses Tool wird im GCode benutzt
			END_IF
 		END_FOR
		
		stGCodeRef.fbLimitCuboid.M_SetDimension(alrHeaderRParam[120], alrHeaderRParam[121], alrHeaderRParam[122],
												alrHeaderRParam[123], alrHeaderRParam[124], alrHeaderRParam[125]);
		
		IF nStateAction < 99 THEN
			IF bStop THEN
				nStateAction := 80;
			ELSE
				nStateAction := 2; //weiter zu ZSensorCheck	
			END_IF
		END_IF
		
	2:	//Checken, ob ein Tool verwendet wird, an desse Achse gerade ein ZSensor angebaut ist
		//Wenn ja, dann eine Auforderung zum Abmontieren senden
		//Gleichzeitig wird die Erreichbarkeit der Scaffoldgrenzen der Tools überprüft
		nStateAction := 80;
		IF NOT bStop THEN
			FOR i:= 1 TO GCode.cMaxGCodeTools BY 1 DO
				IF stGCodeRef.aToolTable[i].pMzTool > 0 AND stGCodeRef.aToolTable[i].bIsUsed THEN
					
					stError.ErrorId := stGCodeRef.aToolTable[i].pMzTool^.M_CheckMoveLimitEx(stGCodeRef.fbLimitCuboid);
					IF stError.ErrorId > 0 THEN
						stError.ObjectId := stGCodeRef.aToolTable[i].pMzTool^.P_nObjectID;
						nStateAction := 99;
						EXIT;
					END_IF
				
					IF stGCodeRef.aToolTable[i].pMzTool^.P_bSensorMounted THEN
						stInteractRequest.nObjectId := stGCodeRef.aToolTable[i].pMzTool^.P_nObjectID;
						stInteractRequest.eInteractMessageType := E_InteractMessageType.INTERACTMES_UnmountZSensor;	//Interaction Request
						nStateAction := 3;
						nCyclCounter := 0;
						EXIT;
					END_IF
				END_IF
			END_FOR
		END_IF
		
	3:	//Request wurde abgesendet und Antwort abwarten
		IF bStop THEN
			nStateAction := 80;
			RETURN;
		END_IF
		
		IF stInterResponse.eInteractMessageType = stInteractRequest.eInteractMessageType THEN
			//50 Zyklen warten, damit das Event auch ankommt
			//damit die Abtastzeit beim Client nicht zu niedrig gewählt werden muss
			nCyclCounter := nCyclCounter + 1;
			IF nCyclCounter = 50 THEN
				nStateAction := 4;
			END_IF
			MEMSET(ADR(stInteractRequest),0,SIZEOF(stInteractRequest));
			MEMSET(ADR(stInterResponse),0,SIZEOF(stInterResponse));			
		ELSIF stInterResponse.eInteractMessageType = E_InteractMessageType.INTERACTMES_Cancel THEN
			nStateAction := 5;
			MEMSET(ADR(stInteractRequest),0,SIZEOF(stInteractRequest));
			MEMSET(ADR(stInterResponse),0,SIZEOF(stInterResponse));			
		END_IF
		
	4:	//Response ist angekommen mit positiver Antwort
		nStateAction := 2;	//erneut checken
	
	5:	//Response ist angekommen mit negativer Antwort
		nStateAction := 81;
END_CASE

IF nStateAction = 80 THEN
	//falls die Oberkante des Scaffolds höher ist als die Kollissionshöhe der Workplate, dann diese erhöhen
	IF stGCodeRef.fbLimitCuboid.P_rZMax > afbWorkplate[1].P_rCollHeight THEN
		IF stGCodeRef.pHead^.P_rMaxCollFreeHeight > stGCodeRef.fbLimitCuboid.P_rZMax THEN
			afbWorkplate[1].P_rCollHeight := stGCodeRef.fbLimitCuboid.P_rZMax + 1000; 
		ELSE
			stError.ErrorId := E_ErrorIdGCode.ERRORID_ScaffoldHeightExceeded;
			nStateAction := 99;
		END_IF
	END_IF	
END_IF
END_ACTION

ACTION A_BasicDispense:
//Nur relevant für Hybrid-Dispenser

stError.POUState := nStateAction;

IF nStateAction = 0 THEN //Preparation
	IF bStop THEN
		nStateAction := 80;
	ELSE
		IF stGCodeRef.pCurrentTool = 0 THEN
			stError.ErrorId := E_ErrorIdGCode.ERRORID_NoSelectedTool;
			nStateAction := 99;
		ELSE 
			IF stGCodeRef.pCurrentTool^.P_eObjectType = E_ObjectType.OBJECTTYPE_HybridDispenser THEN
				pHybridDispenser := stGCodeRef.pCurrentTool;
			ELSE
				nStateAction := 99;
				RETURN;
			END_IF
			IF NOT fbItpReadRParams.bBusy THEN
				IF alrRParam[1] >= 1.0 THEN //Preparation? R1=Prepare
					pHybridDispenser^.M_Prepare(FALSE);
					stMethResult := pHybridDispenser^.M_Prepare(TRUE);
					nStateAction := 1;
				ELSE
					nStateAction := 2;
				END_IF
			END_IF
		END_IF
	END_IF
ELSIF nStateAction = 1 THEN //Preparation fertig?
	IF bStop THEN
		nStateAction := 80;
	ELSE
		stMethResult := pHybridDispenser^.M_Prepare(TRUE);
		IF NOT stMethResult.bBusy THEN
			IF stMethResult.bError THEN
				stError.ErrorId := nErrorId := stMethResult.nErrorId;
				nStateAction := 99;
			ELSE
				//Preparing ready
				nStateAction := 2; //weiter zu Start dispensing
			END_IF
		END_IF
	END_IF
END_IF

IF nStateAction = 2 THEN //Start hybrid dispenser and timer
	IF bStop THEN
		nStateAction := 80;
	ELSE
		stGCodeRef.aToolTable[stGCodeRef.sNciToPlc.Tool].bIsInAction1 := TRUE;
		tDelay := LREAL_TO_TIME(alrRParam[2]); //R2=Start break
		timer(IN:=FALSE);
		IF tDelay > T#0S THEN
			timer(IN:=TRUE,PT:=tDelay);
			stGCodeRef.aToolTable[stGCodeRef.sNciToPlc.Tool].tDelayStart := tDelay;
			nStateAction := 3;
		ELSE
			stGCodeRef.aToolTable[stGCodeRef.sNciToPlc.Tool].tDelayStart := T#0s;
			nStateAction := 80;
		END_IF					
		MEMSET(ADR(stActionData),0,SIZEOF(stActionData));
		stActionData.eAction := E_Action.ACTION_BasicDispense;
		stActionData.aParams[1] := 1; //Start
		stError.ErrorId := pHybridDispenser^.M_ExeAction(stActionData);
		IF stError.ErrorId > 0 THEN
			nStateAction := 99;
		END_IF
	END_IF
ELSIF nStateAction = 3 THEN
	IF bStop THEN
		timer(IN:= FALSE);
		pHybridDispenser^.M_CancelAction(E_Action.ACTION_BasicDispense);
		nStateAction := 80;
		RETURN;
	END_IF
	timer();
	IF timer.Q THEN
		timer(IN:= FALSE);		
		nStateAction := 80;
	END_IF
END_IF
END_ACTION

ACTION A_CleanTip:
stError.POUState := nStateAction;

IF fbComplexAction.bError THEN
	stError.ErrorId :=fbComplexAction.nErrorId;
	nStateAction := 99;
	RETURN;
END_IF

CASE nStateAction OF
	0:	//Aktuelles Tool ausgewählt?
		IF stGCodeRef.pCurrentTool = 0 THEN
			stError.ErrorId := E_ErrorIdGCode.ERRORID_NoSelectedTool;
			nStateAction := 99;
		ELSE
			IF NOT fbItpReadRParams.bBusy THEN
				//konfigurierten TipCleaner ermitteln
				pTarget := fbObjectDirectory.M_GetTipCleaner();
				IF pTarget > 0 THEN
					//NCI-Gruppe auflösen
					fbClearGroup(stGCodeRef:= stGCodeRef, bReGearInSlave:= TRUE, bExecute:= TRUE);
					IF NOT fbClearGroup.bBusy THEN
						IF fbClearGroup.bError THEN
							nStateAction := 99;
							stError.ErrorId := fbClearGroup.nErrorId;
						ELSE
							stCurrentPos := pNewTool^.P_stCurrentPosTotal;
							IF bStop THEN
								nStateAction := 80;
							ELSE
								nStateAction := 1;	
							END_IF
						END_IF
						fbClearGroup(stGCodeRef:= stGCodeRef, bExecute:= FALSE);			
					END_IF
				ELSE
					stError.ObjectId := stGCodeRef.pCurrentTool^.P_nObjectID;
					stError.ErrorId := E_ErrorIdCmd.ERRORID_NoTipCleanerConfigured;
					nStateAction := 99;
				END_IF
			END_IF
		END_IF
		
	1:	//Action "CleanTip" ausführen
		IF bStop THEN
			nStateAction := 80;
			RETURN;
		END_IF
		MEMSET(ADR(stActionData),0,SIZEOF(stActionData));
		stActionData.eAction := E_Action.ACTION_CleanTip;
		stActionData.nObject := stGCodeRef.pCurrentTool^.P_nObjectID;
		stActionData.nTarget := pTarget^.P_nObjectID;
		stActionData.aParams[1] := LREAL_TO_DINT(alrRParam[1]);
		stActionData.aParams[2] := LREAL_TO_DINT(alrRParam[2]);
		stActionData.aParams[3] := LREAL_TO_DINT(alrRParam[3]);
		stActionData.aParams[4] := LREAL_TO_DINT(alrRParam[4]);

		stError.ErrorId := fbComplexAction.M_ExeAction(stActionData);
		IF stError.ErrorId > 0 THEN
			nStateAction := 99;
		ELSE
			nStateAction := 2;	
		END_IF
		
